// TIA Portal V16 program export: 0 tag tables, 0 data types, 94 data blocks, 48 code blocks (in call order from the OBs), 0 instance data blocks

DATA_BLOCK "DBl_SCALE_CS_1"
{ S7_Optimized_Access := 'FALSE' }
VERSION : 0.1
   STRUCT 
      Data { S7_SetPoint := 'False'} : "UDT_SIWA_CS";
   END_STRUCT;


BEGIN

END_DATA_BLOCK

DATA_BLOCK "DBl_SCALE_CS_2"
{ S7_Optimized_Access := 'FALSE' }
VERSION : 0.1
   STRUCT 
      Data { S7_SetPoint := 'False'} : "UDT_SIWA_CS";
   END_STRUCT;


BEGIN

END_DATA_BLOCK

DATA_BLOCK "DB_DateTime"
{ S7_Optimized_Access := 'FALSE' }
VERSION : 0.1
NON_RETAIN
   STRUCT 
      TimeOfDay_PLC : Time_Of_Day;
      Date_PLC : Date;
      DateTime_PLC : Date_And_Time;
      stReadDataTime_PLC : Int;
   END_STRUCT;


BEGIN
   TimeOfDay_PLC := TOD#16:14:12.371;
   Date_PLC := D#2021-11-15;
   DateTime_PLC := DT#2021-11-15-16:14:12.374;
   stReadDataTime_PLC := 0;

END_DATA_BLOCK

DATA_BLOCK "DB_Global"
{ S7_Optimized_Access := 'FALSE' }
VERSION : 0.1
NON_RETAIN
// 2. GLOBAL DATA (Pure Data only)
   STRUCT 
      Sys { ExternalAccessible := 'False'; ExternalVisible := 'False'; ExternalWritable := 'False'; S7_SetPoint := 'False'} : "UDT_Sys_Info";
      c_stDI_Mode { ExternalAccessible := 'False'; ExternalVisible := 'False'; ExternalWritable := 'False'} : Struct
         None { ExternalAccessible := 'False'; ExternalVisible := 'False'; ExternalWritable := 'False'} : Int;
         NOpen { ExternalAccessible := 'False'; ExternalVisible := 'False'; ExternalWritable := 'False'} : Int;
         NClose { ExternalAccessible := 'False'; ExternalVisible := 'False'; ExternalWritable := 'False'} : Int;
         Disabled { ExternalAccessible := 'False'; ExternalVisible := 'False'; ExternalWritable := 'False'} : Int;
      END_STRUCT;
   END_STRUCT;


BEGIN
   Sys.CycleTime_ms_INT := 10;
   Sys.CycleTime_ms_REAL := 10.0;
   c_stDI_Mode.NOpen := 1;
   c_stDI_Mode.NClose := 2;
   c_stDI_Mode.Disabled := 3;

END_DATA_BLOCK

DATA_BLOCK "DB_Log_Buffer"
{ S7_Optimized_Access := 'FALSE' }
VERSION : 0.1
   STRUCT 
      Write_Index : Int;   // Указатель для ПЛК (куда пишем следующую запись)
      Read_Index : Int;   // Указатель для Python/1C (что считано)
      Buffer : Array[0..1999] of "UDT_Log_Record";   // Кольцевой буфер на 500 записей
   END_STRUCT;


BEGIN
   Write_Index := 0;
   Read_Index := 0;

END_DATA_BLOCK

DATA_BLOCK "DB_MAP"
{ S7_Optimized_Access := 'FALSE' }
VERSION : 0.1
NON_RETAIN
   STRUCT 
      HMI_Whouse : Struct
         TRN { S7_SetPoint := 'False'} : "UDT_HMI_Whouse";
         POL { S7_SetPoint := 'False'} : "UDT_HMI_Whouse";
         BUL { S7_SetPoint := 'False'} : "UDT_HMI_Whouse";
         MOL { S7_SetPoint := 'False'} : "UDT_HMI_Whouse";
      END_STRUCT;
      HMI_TRN_SmalTank { S7_SetPoint := 'False'} : Array[1..3] of "UDT_HMI_SmallTank";
      HMI_POL_SmalTank { S7_SetPoint := 'False'} : Array[1..10] of "UDT_HMI_SmallTank";
      HMI_BUL_SmalTank { S7_SetPoint := 'False'} : Array[1..4] of "UDT_HMI_SmallTank";
      HMI_MOL_SmalTank { S7_SetPoint := 'False'} : Array[1..12] of "UDT_HMI_SmallTank";
      Scale_CS_1 : "UDT_Siwarex_Core";
      Scale_CS_2 : "UDT_Siwarex_Core";
   END_STRUCT;


BEGIN

END_DATA_BLOCK

DATA_BLOCK "DB_Wh_BUL"
{ S7_Optimized_Access := 'FALSE' }
VERSION : 0.1
   STRUCT 
      Tank : Array[1..4] of "UDT_Tank_Full";
   END_STRUCT;


BEGIN

END_DATA_BLOCK

DATA_BLOCK "DB_Wh_MOL"
{ S7_Optimized_Access := 'FALSE' }
VERSION : 0.1
   STRUCT 
      Tank : Array[1..10] of "UDT_Tank_Full";
   END_STRUCT;


BEGIN

END_DATA_BLOCK

DATA_BLOCK "DB_Wh_POL"
{ S7_Optimized_Access := 'FALSE' }
VERSION : 0.1
   STRUCT 
      Tank : Array[1..10] of "UDT_Tank_Full";
   END_STRUCT;


BEGIN

END_DATA_BLOCK

DATA_BLOCK "DB_Wh_TRN"
{ S7_Optimized_Access := 'FALSE' }
VERSION : 0.1
   STRUCT 
      HMI_Word_spare : DWord;
      Tank : Array[1..3] of "UDT_Tank_Full";
   END_STRUCT;


BEGIN

END_DATA_BLOCK

DATA_BLOCK "Total_DB"
{ S7_Optimized_Access := 'FALSE' }
VERSION : 0.1
NON_RETAIN
   STRUCT 
      Total_Reset_HMI : Bool;
      Restart_PLC : Bool;
   END_STRUCT;


BEGIN
   Total_Reset_HMI := FALSE;
   Restart_PLC := FALSE;

END_DATA_BLOCK

DATA_BLOCK "iDB_BUL_Tank_Log_1"
{ S7_Optimized_Access := 'FALSE' }
AUTHOR : Gemini
FAMILY : Archive
VERSION : 1.2
NON_RETAIN
"FB_Tank_Logic"

BEGIN

END_DATA_BLOCK

DATA_BLOCK "iDB_BUL_Tank_Log_2"
{ S7_Optimized_Access := 'FALSE' }
AUTHOR : Gemini
FAMILY : Archive
VERSION : 1.2
NON_RETAIN
"FB_Tank_Logic"

BEGIN

END_DATA_BLOCK

DATA_BLOCK "iDB_BUL_Tank_Log_3"
{ S7_Optimized_Access := 'FALSE' }
AUTHOR : Gemini
FAMILY : Archive
VERSION : 1.2
NON_RETAIN
"FB_Tank_Logic"

BEGIN

END_DATA_BLOCK

DATA_BLOCK "iDB_BUL_Tank_Log_4"
{ S7_Optimized_Access := 'FALSE' }
AUTHOR : Gemini
FAMILY : Archive
VERSION : 1.2
NON_RETAIN
"FB_Tank_Logic"

BEGIN

END_DATA_BLOCK

DATA_BLOCK "iDB_MOL_Tank_Log_1"
{ S7_Optimized_Access := 'FALSE' }
AUTHOR : Gemini
FAMILY : Archive
VERSION : 1.2
NON_RETAIN
"FB_Tank_Logic"

BEGIN

END_DATA_BLOCK

DATA_BLOCK "iDB_MOL_Tank_Log_10"
{ S7_Optimized_Access := 'FALSE' }
AUTHOR : Gemini
FAMILY : Archive
VERSION : 1.2
NON_RETAIN
"FB_Tank_Logic"

BEGIN

END_DATA_BLOCK

DATA_BLOCK "iDB_MOL_Tank_Log_11"
{ S7_Optimized_Access := 'FALSE' }
AUTHOR : Gemini
FAMILY : Archive
VERSION : 1.2
NON_RETAIN
"FB_Tank_Logic"

BEGIN

END_DATA_BLOCK

DATA_BLOCK "iDB_MOL_Tank_Log_12"
{ S7_Optimized_Access := 'FALSE' }
AUTHOR : Gemini
FAMILY : Archive
VERSION : 1.2
NON_RETAIN
"FB_Tank_Logic"

BEGIN

END_DATA_BLOCK

DATA_BLOCK "iDB_MOL_Tank_Log_2"
{ S7_Optimized_Access := 'FALSE' }
AUTHOR : Gemini
FAMILY : Archive
VERSION : 1.2
NON_RETAIN
"FB_Tank_Logic"

BEGIN

END_DATA_BLOCK

DATA_BLOCK "iDB_MOL_Tank_Log_3"
{ S7_Optimized_Access := 'FALSE' }
AUTHOR : Gemini
FAMILY : Archive
VERSION : 1.2
NON_RETAIN
"FB_Tank_Logic"

BEGIN

END_DATA_BLOCK

DATA_BLOCK "iDB_MOL_Tank_Log_4"
{ S7_Optimized_Access := 'FALSE' }
AUTHOR : Gemini
FAMILY : Archive
VERSION : 1.2
NON_RETAIN
"FB_Tank_Logic"

BEGIN

END_DATA_BLOCK

DATA_BLOCK "iDB_MOL_Tank_Log_5"
{ S7_Optimized_Access := 'FALSE' }
AUTHOR : Gemini
FAMILY : Archive
VERSION : 1.2
NON_RETAIN
"FB_Tank_Logic"

BEGIN

END_DATA_BLOCK

DATA_BLOCK "iDB_MOL_Tank_Log_6"
{ S7_Optimized_Access := 'FALSE' }
AUTHOR : Gemini
FAMILY : Archive
VERSION : 1.2
NON_RETAIN
"FB_Tank_Logic"

BEGIN

END_DATA_BLOCK

DATA_BLOCK "iDB_MOL_Tank_Log_7"
{ S7_Optimized_Access := 'FALSE' }
AUTHOR : Gemini
FAMILY : Archive
VERSION : 1.2
NON_RETAIN
"FB_Tank_Logic"

BEGIN

END_DATA_BLOCK

DATA_BLOCK "iDB_MOL_Tank_Log_8"
{ S7_Optimized_Access := 'FALSE' }
AUTHOR : Gemini
FAMILY : Archive
VERSION : 1.2
NON_RETAIN
"FB_Tank_Logic"

BEGIN

END_DATA_BLOCK

DATA_BLOCK "iDB_MOL_Tank_Log_9"
{ S7_Optimized_Access := 'FALSE' }
AUTHOR : Gemini
FAMILY : Archive
VERSION : 1.2
NON_RETAIN
"FB_Tank_Logic"

BEGIN

END_DATA_BLOCK

DATA_BLOCK "iDB_POL_Tank_Log_1"
{ S7_Optimized_Access := 'FALSE' }
AUTHOR : Gemini
FAMILY : Archive
VERSION : 1.2
"FB_Tank_Logic"

BEGIN

END_DATA_BLOCK

DATA_BLOCK "iDB_POL_Tank_Log_10"
{ S7_Optimized_Access := 'FALSE' }
AUTHOR : Gemini
FAMILY : Archive
VERSION : 1.2
NON_RETAIN
"FB_Tank_Logic"

BEGIN

END_DATA_BLOCK

DATA_BLOCK "iDB_POL_Tank_Log_3"
{ S7_Optimized_Access := 'FALSE' }
AUTHOR : Gemini
FAMILY : Archive
VERSION : 1.2
"FB_Tank_Logic"

BEGIN

END_DATA_BLOCK

DATA_BLOCK "iDB_POL_Tank_Log_4"
{ S7_Optimized_Access := 'FALSE' }
AUTHOR : Gemini
FAMILY : Archive
VERSION : 1.2
"FB_Tank_Logic"

BEGIN

END_DATA_BLOCK

DATA_BLOCK "iDB_POL_Tank_Log_5"
{ S7_Optimized_Access := 'FALSE' }
AUTHOR : Gemini
FAMILY : Archive
VERSION : 1.2
"FB_Tank_Logic"

BEGIN

END_DATA_BLOCK

DATA_BLOCK "iDB_POL_Tank_Log_6"
{ S7_Optimized_Access := 'FALSE' }
AUTHOR : Gemini
FAMILY : Archive
VERSION : 1.2
"FB_Tank_Logic"

BEGIN

END_DATA_BLOCK

DATA_BLOCK "iDB_POL_Tank_Log_7"
{ S7_Optimized_Access := 'FALSE' }
AUTHOR : Gemini
FAMILY : Archive
VERSION : 1.2
NON_RETAIN
"FB_Tank_Logic"

BEGIN

END_DATA_BLOCK

DATA_BLOCK "iDB_POL_Tank_Log_8"
{ S7_Optimized_Access := 'FALSE' }
AUTHOR : Gemini
FAMILY : Archive
VERSION : 1.2
NON_RETAIN
"FB_Tank_Logic"

BEGIN

END_DATA_BLOCK

DATA_BLOCK "iDB_POL_Tank_Log_9"
{ S7_Optimized_Access := 'FALSE' }
AUTHOR : Gemini
FAMILY : Archive
VERSION : 1.2
NON_RETAIN
"FB_Tank_Logic"

BEGIN

END_DATA_BLOCK

DATA_BLOCK "iDB_TRN_Tank_Log_1"
{ S7_Optimized_Access := 'FALSE' }
AUTHOR : Gemini
FAMILY : Archive
VERSION : 1.2
NON_RETAIN
"FB_Tank_Logic"

BEGIN

END_DATA_BLOCK

DATA_BLOCK "iDB_TRN_Tank_Log_2"
{ S7_Optimized_Access := 'FALSE' }
AUTHOR : Gemini
FAMILY : Archive
VERSION : 1.2
NON_RETAIN
"FB_Tank_Logic"

BEGIN

END_DATA_BLOCK

DATA_BLOCK "iDB_TRN_Tank_Log_3"
{ S7_Optimized_Access := 'FALSE' }
AUTHOR : Gemini
FAMILY : Archive
VERSION : 1.2
NON_RETAIN
"FB_Tank_Logic"

BEGIN

END_DATA_BLOCK

DATA_BLOCK "iDB_Time_Trigger"
{ S7_Optimized_Access := 'FALSE' }
AUTHOR : S7A_Lib
FAMILY : Archive
VERSION : 1.1
"FB_Time_Trigger"

BEGIN

END_DATA_BLOCK

DATA_BLOCK "Pol_sklad_db"
{ S7_Optimized_Access := 'FALSE' }
VERSION : 0.1
   STRUCT 
      Pol_p : Real;
      Eror_pol_p : DWord;
      S_pol : Real;
      Weigt : Real;
      Densyty : Real;
      "1_pol" : Struct
         Weight_db : Real;
         Weight_zero : Real;
         Weight_Formula_W_T : Real;
         Visible : Bool;
         p_zero : Real;
         p_weight : Real;
         Zero_but : Bool;
         Weight_but : Bool;
         S : Real;
         Densyty : Real;
         Korect : Bool;
      END_STRUCT;
      "2_pol" : Struct
         Weight_db : Real;
         Weight_zero : Real;
         Weight_Formula_W_T : Real;
         Visible : Bool;
         p_zero : Real;
         p_weight : Real;
         Zero_but : Bool;
         Weight_but : Bool;
         S : Real;
         Densyty : Real;
         Korect : Bool;
      END_STRUCT;
      "3_pol" : Struct
         Weight_db : Real;
         Weight_zero : Real;
         Weight_Formula_W_T : Real;
         Visible : Bool;
         p_zero : Real;
         p_weight : Real;
         Zero_but : Bool;
         Weight_but : Bool;
         S : Real;
         Densyty : Real;
         Korect : Bool;
      END_STRUCT;
      "4_pol" : Struct
         Weight_db : Real;
         Weight_zero : Real;
         Weight_Formula_W_T : Real;
         Visible : Bool;
         p_zero : Real;
         p_weight : Real;
         Zero_but : Bool;
         Weight_but : Bool;
         S : Real;
         Densyty : Real;
         Korect : Bool;
      END_STRUCT;
      "5_pol" : Struct
         Weight_db : Real;
         Weight_zero : Real;
         Weight_Formula_W_T : Real;
         Visible : Bool;
         p_zero : Real;
         p_weight : Real;
         Zero_but : Bool;
         Weight_but : Bool;
         S : Real;
         Densyty : Real;
         Korect : Bool;
      END_STRUCT;
      "6_pol" : Struct
         Weight_db : Real;
         Weight_zero : Real;
         Weight_Formula_W_T : Real;
         Visible : Bool;
         p_zero : Real;
         p_weight : Real;
         Zero_but : Bool;
         Weight_but : Bool;
         S : Real;
         Densyty : Real;
         Korect : Bool;
      END_STRUCT;
      "7_pol" : Struct
         Weight_db : Real;
         Weight_zero : Real;
         Weight_Formula_W_T : Real;
         Visible : Bool;
         p_zero : Real;
         p_weight : Real;
         Zero_but : Bool;
         Weight_but : Bool;
         S : Real;
         Densyty : Real;
         Korect : Bool;
      END_STRUCT;
      "8_pol" : Struct
         Weight_db : Real;
         Weight_zero : Real;
         Weight_Formula_W_T : Real;
         Visible : Bool;
         p_zero : Real;
         p_weight : Real;
         Zero_but : Bool;
         Weight_but : Bool;
         S : Real;
         Densyty : Real;
         Korect : Bool;
      END_STRUCT;
      "9_pol" : Struct
         Weight_db : Real;
         Weight_zero : Real;
         Weight_Formula_W_T : Real;
         Visible : Bool;
         p_zero : Real;
         p_weight : Real;
         Zero_but : Bool;
         Weight_but : Bool;
         S : Real;
         Densyty : Real;
         Korect : Bool;
      END_STRUCT;
      "10_pol" : Struct
         Weight_db : Real;
         Weight_zero : Real;
         Weight_Formula_W_T : Real;
         Visible : Bool;
         p_zero : Real;
         p_weight : Real;
         Zero_but : Bool;
         Weight_but : Bool;
         S : Real;
         Densyty : Real;
         Korect : Bool;
      END_STRUCT;
   END_STRUCT;


BEGIN
   Pol_p := 1.149812;
   Eror_pol_p := 16#0000_0000;
   S_pol := 6.819987;
   Weigt := 79.9358;
   Densyty := 1.35;
   "1_pol".Weight_db := 0.0;
   "1_pol".Weight_zero := 0.0;
   "1_pol".Weight_Formula_W_T := 81.81128;
   "1_pol".Visible := TRUE;
   "1_pol".p_zero := 0.0;
   "1_pol".p_weight := 0.0;
   "1_pol".Zero_but := FALSE;
   "1_pol".Weight_but := FALSE;
   "1_pol".S := 6.98;
   "1_pol".Densyty := 1.35;
   "1_pol".Korect := FALSE;
   "2_pol".Weight_db := 19.52373;
   "2_pol".Weight_zero := 0.0;
   "2_pol".Weight_Formula_W_T := 78.76387;
   "2_pol".Visible := FALSE;
   "2_pol".p_zero := 0.0;
   "2_pol".p_weight := 0.2850116;
   "2_pol".Zero_but := FALSE;
   "2_pol".Weight_but := FALSE;
   "2_pol".S := 6.72;
   "2_pol".Densyty := 1.35;
   "2_pol".Korect := FALSE;
   "3_pol".Weight_db := 0.0;
   "3_pol".Weight_zero := 0.0;
   "3_pol".Weight_Formula_W_T := 78.52945;
   "3_pol".Visible := FALSE;
   "3_pol".p_zero := 0.0;
   "3_pol".p_weight := 0.0;
   "3_pol".Zero_but := FALSE;
   "3_pol".Weight_but := FALSE;
   "3_pol".S := 6.7;
   "3_pol".Densyty := 1.35;
   "3_pol".Korect := FALSE;
   "4_pol".Weight_db := 73.68473;
   "4_pol".Weight_zero := 0.0;
   "4_pol".Weight_Formula_W_T := 78.76387;
   "4_pol".Visible := FALSE;
   "4_pol".p_zero := 0.0;
   "4_pol".p_weight := 1.075665;
   "4_pol".Zero_but := FALSE;
   "4_pol".Weight_but := FALSE;
   "4_pol".S := 6.72;
   "4_pol".Densyty := 1.35;
   "4_pol".Korect := FALSE;
   "5_pol".Weight_db := 24.61529;
   "5_pol".Weight_zero := 0.0;
   "5_pol".Weight_Formula_W_T := 77.55404;
   "5_pol".Visible := FALSE;
   "5_pol".p_zero := 0.0;
   "5_pol".p_weight := 0.364945;
   "5_pol".Zero_but := FALSE;
   "5_pol".Weight_but := FALSE;
   "5_pol".S := 6.61678;
   "5_pol".Densyty := 1.35;
   "5_pol".Korect := FALSE;
   "6_pol".Weight_db := 49.182;
   "6_pol".Weight_zero := 0.0;
   "6_pol".Weight_Formula_W_T := 78.64666;
   "6_pol".Visible := FALSE;
   "6_pol".p_zero := 0.0;
   "6_pol".p_weight := 0.7190394;
   "6_pol".Zero_but := FALSE;
   "6_pol".Weight_but := FALSE;
   "6_pol".S := 6.71;
   "6_pol".Densyty := 1.35;
   "6_pol".Korect := FALSE;
   "7_pol".Weight_db := 123.4003;
   "7_pol".Weight_zero := 0.0;
   "7_pol".Weight_Formula_W_T := 78.64666;
   "7_pol".Visible := FALSE;
   "7_pol".p_zero := 0.0;
   "7_pol".p_weight := 1.804109;
   "7_pol".Zero_but := FALSE;
   "7_pol".Weight_but := FALSE;
   "7_pol".S := 6.71;
   "7_pol".Densyty := 1.35;
   "7_pol".Korect := FALSE;
   "8_pol".Weight_db := -0.2724785;
   "8_pol".Weight_zero := 0.4211032;
   "8_pol".Weight_Formula_W_T := 78.74628;
   "8_pol".Visible := FALSE;
   "8_pol".p_zero := 0.006148727;
   "8_pol".p_weight := 0.002170139;
   "8_pol".Zero_but := FALSE;
   "8_pol".Weight_but := FALSE;
   "8_pol".S := 6.7185;
   "8_pol".Densyty := 1.35;
   "8_pol".Korect := FALSE;
   "9_pol".Weight_db := 126.8467;
   "9_pol".Weight_zero := 0.0;
   "9_pol".Weight_Formula_W_T := 78.97484;
   "9_pol".Visible := FALSE;
   "9_pol".p_zero := 0.0;
   "9_pol".p_weight := 1.846788;
   "9_pol".Zero_but := FALSE;
   "9_pol".Weight_but := FALSE;
   "9_pol".S := 6.738;
   "9_pol".Densyty := 1.35;
   "9_pol".Korect := FALSE;
   "10_pol".Weight_db := 27.88432;
   "10_pol".Weight_zero := 0.0;
   "10_pol".Weight_Formula_W_T := 77.55404;
   "10_pol".Visible := TRUE;
   "10_pol".p_zero := 0.0;
   "10_pol".p_weight := 0.4134114;
   "10_pol".Zero_but := FALSE;
   "10_pol".Weight_but := FALSE;
   "10_pol".S := 6.61678;
   "10_pol".Densyty := 1.35;
   "10_pol".Korect := FALSE;

END_DATA_BLOCK

DATA_BLOCK "iDB_Map_Siwarex_Core"
{ S7_Optimized_Access := 'FALSE' }
AUTHOR : S7C_Lib
FAMILY : Analog
VERSION : 1.4
"FB_Map_Siwarex_Core"

BEGIN

END_DATA_BLOCK

DATA_BLOCK "iFB_Map_Siwarex_Core"
{ S7_Optimized_Access := 'FALSE' }
AUTHOR : S7C_Lib
FAMILY : Analog
VERSION : 1.4
"FB_Map_Siwarex_Core"

BEGIN

END_DATA_BLOCK

DATA_BLOCK "MaxLevels"
{ S7_Optimized_Access := 'FALSE' }
VERSION : 0.1
   STRUCT 
      MaxLevel_Tank_1 : Real;
      MaxLevel_Tank_2 : Real;
      MaxLevel_Tank_3 : Real;
      MaxLevel_Tank_4 : Real;
      MaxLevel_Tank_5 : Real;
      MaxLevel_Tank_6 : Real;
      MaxLevel_Tank_7 : Real;
      MaxLevel_Tank_8 : Real;
      MaxLevel_Tank_9 : Real;
      MaxLevel_Tank_10 : Real;
      MaxLevel_Tank_11 : Real;
      MaxLevel_Tank_12 : Real;
      MaxLevel_Tank_13 : Real;
      MaxLevel_Tank_14 : Real;
   END_STRUCT;


BEGIN
   MaxLevel_Tank_1 := 15.0;
   MaxLevel_Tank_2 := 15.0;
   MaxLevel_Tank_3 := 15.0;
   MaxLevel_Tank_4 := 15.0;
   MaxLevel_Tank_5 := 15.0;
   MaxLevel_Tank_6 := 15.0;
   MaxLevel_Tank_7 := 15.0;
   MaxLevel_Tank_8 := 15.0;
   MaxLevel_Tank_9 := 15.0;
   MaxLevel_Tank_10 := 15.0;
   MaxLevel_Tank_11 := 13.0;
   MaxLevel_Tank_12 := 13.0;
   MaxLevel_Tank_13 := 13.0;
   MaxLevel_Tank_14 := 13.0;

END_DATA_BLOCK

DATA_BLOCK "DB_SCALE_CS_1"
{ S7_Optimized_Access := 'FALSE' }
VERSION : 0.0
"UDT_SIWA_CS"

BEGIN
   i_DB_Lenght := 222;
   i_MaxLifeBitCyc := 500;
   i_SFC_ERR_C := 16#0000;
   i_CMD_INPUT := 230;
   bo_CMD_TRIGGER := TRUE;
   bo_CMD_IN_PROGRESS := TRUE;
   bo_CMD_FINISHED_OK := FALSE;
   bo_CMD_ERR := FALSE;
   b_CMD_ERR_CODE := 16#00;
   i_PRESET_TARE := 0;
   b_SELECT_PROC_VAL := 16#00;
   b_SELECTED_PROC_VAL := 16#00;
   i_PROCESS_VALUE := 215;
   b_INFO_REFRESH_COUNT := 16#5A;
   w_SCALE_STATUS := 16#00C0;
   b_OPR_ERR_MSG := 16#00;
   bo_FB_ERR := FALSE;
   b_FB_ERR_CODE := 16#00;
   bo_START_UP_IN_PROGRESS := FALSE;
   w_DB_RES92 := 16#0000;
   w_DB_RES93 := 16#0000;
   w_DB_RES94 := 16#0000;
   w_DB_RES95 := 16#0000;
   w_DB_RES96 := 16#0000;
   w_DB_RES97 := 16#0000;
   w_INT_USE := 16#0000;
   s_JUST_DAT.w_CALIB_DIGITS0 := 16#0000;
   s_JUST_DAT.w_CALIB_DIGITS1 := 16#EA60;
   s_JUST_DAT.w_CALIB_DIGITS2 := 16#0000;
   s_JUST_DAT.i_CALIB_WEIGHT1 := 2000;
   s_JUST_DAT.i_CALIB_WEIGHT2 := 0;
   s_JUST_DAT.b_SIGNAL_RANGE := 16#02;
   s_JUST_DAT.b_FILT_TYPE := 16#00;
   s_JUST_DAT.b_FILT_FREQ := 16#04;
   s_JUST_DAT.b_FILT_DEPTH := 16#0F;
   s_JUST_DAT.s_SCALE_ID := 'SIWAREX XX';
   s_JUST_DAT.i_MIN_WR := 20;
   s_JUST_DAT.i_MAX_WR := 2000;
   s_JUST_DAT.i_INCREMENT_WR := 1;
   s_JUST_DAT.i_WEIGHT_ST_STILL := 10;
   s_JUST_DAT.t_TIME_ST_STILL1 := T#1S;
   s_JUST_DAT.b_DEC_POINT := 16#02;
   s_JUST_DAT.b_ZERO_NEG_VALUE := 16#01;
   s_JUST_DAT.b_ZERO_POS_VALUE := 16#03;
   s_JUST_DAT.b_TARA_MAX := 16#64;
   s_JUST_DAT.i_Reserve := 0;
   s_JUST_DAT.s_LEGAL_TRADE := '----';
   s_JUST_DAT.s_WEGHT_UNIT := 'kg  ';
   s_LIMIT_PARA.i_LIMIT1_ON := 400;
   s_LIMIT_PARA.i_LIMIT1_OFF := 220;
   s_LIMIT_PARA.i_LIMIT2_ON := 1000;
   s_LIMIT_PARA.i_LIMIT2_OFF := 980;
   s_LIMIT_PARA.bo_LIMIT1_PARA := FALSE;
   s_LIMIT_PARA.bo_LIMIT2_PARA := FALSE;
   s_LIMIT_PARA.b_Reserve := 16#00;
   s_MODUL_INFO_DATA.s_MODUL_NAME := 'SIWAREX CS';
   s_MODUL_INFO_DATA.s_ORDER_NUM := '7MH4910-0AA01$00$00$00$00   ';
   s_MODUL_INFO_DATA.w_VERSION_HW := 16#0005;
   s_MODUL_INFO_DATA.s_VERSION_FW := 'V1.5';
   s_MODUL_INFO_DATA.w_CRC_CHECK := 16#0897;
   s_TARE_CONTROL.i_TARE_VALUE := 0;
   s_INTERNAL_PROC_VAL.w_CRC_CHECK := 16#0000;
   s_INTERNAL_PROC_VAL.b_Reserve := 16#00;
   s_INTERNAL_PROC_VAL.bo_PRESET_TARA := FALSE;
   s_INTERNAL_PROC_VAL.d_TARA_X_100 := 0;
   s_INTERNAL_PROC_VAL.d_ZERO_X_100 := 0;
   s_PROCESS_VALUES.w_CRC_CHECK := 16#4732;
   s_PROCESS_VALUES.bo_STA_WRI_PROT := FALSE;
   s_PROCESS_VALUES.bo_STA_WR_MIN := FALSE;
   s_PROCESS_VALUES.bo_STA_Reserve1 := FALSE;
   s_PROCESS_VALUES.bo_STA_Reserve2 := FALSE;
   s_PROCESS_VALUES.bo_STA_Reserve3 := FALSE;
   s_PROCESS_VALUES.bo_STA_Reserve4 := FALSE;
   s_PROCESS_VALUES.bo_STA_Reserve5 := FALSE;
   s_PROCESS_VALUES.bo_STA_ERROR_ON := FALSE;
   s_PROCESS_VALUES.bo_STA_LIMIT1_ON := FALSE;
   s_PROCESS_VALUES.bo_STA_LIMIT2_ON := FALSE;
   s_PROCESS_VALUES.bo_STA_TARED := FALSE;
   s_PROCESS_VALUES.bo_STA_TARED_BY_MANUAL := FALSE;
   s_PROCESS_VALUES.bo_STA_MAX_9E := FALSE;
   s_PROCESS_VALUES.bo_STA_025_D_ZERO := FALSE;
   s_PROCESS_VALUES.bo_STA_ST_STAND_SCALE_ON := TRUE;
   s_PROCESS_VALUES.bo_STA_SCALE_CALIBRATED := TRUE;
   s_PROCESS_VALUES.b_OPR_ERR_MSG := 16#00;
   s_PROCESS_VALUES.b_Reserve := 16#00;
   s_PROCESS_VALUES.i_GROSS_WEIGHT_PROC := 217;
   s_PROCESS_VALUES.i_NET_WEIGHT_PROC := 217;
   s_PROCESS_VALUES.i_TARE_WEIGHT_PROC := 0;
   s_PROCESS_VALUES.i_GROSS_NET_VALUE := 215;
   s_PROCESS_VALUES.d_GROSS_NET_VALUE_10X := 2175;
   s_PROCESS_VALUES.i_TARE_VALUE := 0;
   s_PROCESS_VALUES.i_ADC_DIGIT := 8980;
   s_PROCESS_VALUES.i_ADC_DIGIT_FILTER := 8982;
   s_PROCESS_VALUES.s_WEIGHT_ASCII := 'B      215kg  ';
   s_PROCESS_VALUES.i_MILISEC := 180;
   s_PROCESS_VALUES.b_SECONDS := 16#2A;
   s_PROCESS_VALUES.b_MINUTE := 16#39;
   s_PROCESS_VALUES.i_HOURS := 57;
   i_DB_Lenght1 := 222;

END_DATA_BLOCK

DATA_BLOCK "DB_SCALE_CS_2"
{ S7_Optimized_Access := 'FALSE' }
VERSION : 0.0
"UDT_SIWA_CS"

BEGIN
   i_DB_Lenght := 222;
   i_MaxLifeBitCyc := 500;
   i_SFC_ERR_C := 16#0000;
   i_CMD_INPUT := 230;
   bo_CMD_TRIGGER := TRUE;
   bo_CMD_IN_PROGRESS := TRUE;
   bo_CMD_FINISHED_OK := FALSE;
   bo_CMD_ERR := FALSE;
   b_CMD_ERR_CODE := 16#00;
   i_PRESET_TARE := 0;
   b_SELECT_PROC_VAL := 16#00;
   b_SELECTED_PROC_VAL := 16#00;
   i_PROCESS_VALUE := -25;
   b_INFO_REFRESH_COUNT := 16#07;
   w_SCALE_STATUS := 16#02C0;
   b_OPR_ERR_MSG := 16#00;
   bo_FB_ERR := FALSE;
   b_FB_ERR_CODE := 16#00;
   bo_START_UP_IN_PROGRESS := FALSE;
   w_DB_RES92 := 16#0000;
   w_DB_RES93 := 16#0000;
   w_DB_RES94 := 16#0000;
   w_DB_RES95 := 16#0000;
   w_DB_RES96 := 16#0000;
   w_DB_RES97 := 16#0000;
   w_INT_USE := 16#0000;
   s_JUST_DAT.w_CALIB_DIGITS0 := 16#0000;
   s_JUST_DAT.w_CALIB_DIGITS1 := 16#EA60;
   s_JUST_DAT.w_CALIB_DIGITS2 := 16#0000;
   s_JUST_DAT.i_CALIB_WEIGHT1 := 2000;
   s_JUST_DAT.i_CALIB_WEIGHT2 := 0;
   s_JUST_DAT.b_SIGNAL_RANGE := 16#02;
   s_JUST_DAT.b_FILT_TYPE := 16#00;
   s_JUST_DAT.b_FILT_FREQ := 16#04;
   s_JUST_DAT.b_FILT_DEPTH := 16#0F;
   s_JUST_DAT.s_SCALE_ID := 'SIWAREX XX';
   s_JUST_DAT.i_MIN_WR := 20;
   s_JUST_DAT.i_MAX_WR := 2000;
   s_JUST_DAT.i_INCREMENT_WR := 1;
   s_JUST_DAT.i_WEIGHT_ST_STILL := 10;
   s_JUST_DAT.t_TIME_ST_STILL1 := T#1S;
   s_JUST_DAT.b_DEC_POINT := 16#02;
   s_JUST_DAT.b_ZERO_NEG_VALUE := 16#01;
   s_JUST_DAT.b_ZERO_POS_VALUE := 16#03;
   s_JUST_DAT.b_TARA_MAX := 16#64;
   s_JUST_DAT.i_Reserve := 0;
   s_JUST_DAT.s_LEGAL_TRADE := '----';
   s_JUST_DAT.s_WEGHT_UNIT := 'kg  ';
   s_LIMIT_PARA.i_LIMIT1_ON := 400;
   s_LIMIT_PARA.i_LIMIT1_OFF := 220;
   s_LIMIT_PARA.i_LIMIT2_ON := 1000;
   s_LIMIT_PARA.i_LIMIT2_OFF := 980;
   s_LIMIT_PARA.bo_LIMIT1_PARA := FALSE;
   s_LIMIT_PARA.bo_LIMIT2_PARA := FALSE;
   s_LIMIT_PARA.b_Reserve := 16#00;
   s_MODUL_INFO_DATA.s_MODUL_NAME := 'SIWAREX CS';
   s_MODUL_INFO_DATA.s_ORDER_NUM := '7MH4910-0AA01$00$00$00$00   ';
   s_MODUL_INFO_DATA.w_VERSION_HW := 16#0005;
   s_MODUL_INFO_DATA.s_VERSION_FW := 'V1.5';
   s_MODUL_INFO_DATA.w_CRC_CHECK := 16#0897;
   s_TARE_CONTROL.i_TARE_VALUE := 0;
   s_INTERNAL_PROC_VAL.w_CRC_CHECK := 16#0000;
   s_INTERNAL_PROC_VAL.b_Reserve := 16#00;
   s_INTERNAL_PROC_VAL.bo_PRESET_TARA := FALSE;
   s_INTERNAL_PROC_VAL.d_TARA_X_100 := 0;
   s_INTERNAL_PROC_VAL.d_ZERO_X_100 := 0;
   s_PROCESS_VALUES.w_CRC_CHECK := 16#9561;
   s_PROCESS_VALUES.bo_STA_WRI_PROT := FALSE;
   s_PROCESS_VALUES.bo_STA_WR_MIN := TRUE;
   s_PROCESS_VALUES.bo_STA_Reserve1 := FALSE;
   s_PROCESS_VALUES.bo_STA_Reserve2 := FALSE;
   s_PROCESS_VALUES.bo_STA_Reserve3 := FALSE;
   s_PROCESS_VALUES.bo_STA_Reserve4 := FALSE;
   s_PROCESS_VALUES.bo_STA_Reserve5 := FALSE;
   s_PROCESS_VALUES.bo_STA_ERROR_ON := FALSE;
   s_PROCESS_VALUES.bo_STA_LIMIT1_ON := FALSE;
   s_PROCESS_VALUES.bo_STA_LIMIT2_ON := FALSE;
   s_PROCESS_VALUES.bo_STA_TARED := FALSE;
   s_PROCESS_VALUES.bo_STA_TARED_BY_MANUAL := FALSE;
   s_PROCESS_VALUES.bo_STA_MAX_9E := FALSE;
   s_PROCESS_VALUES.bo_STA_025_D_ZERO := FALSE;
   s_PROCESS_VALUES.bo_STA_ST_STAND_SCALE_ON := TRUE;
   s_PROCESS_VALUES.bo_STA_SCALE_CALIBRATED := TRUE;
   s_PROCESS_VALUES.b_OPR_ERR_MSG := 16#00;
   s_PROCESS_VALUES.b_Reserve := 16#00;
   s_PROCESS_VALUES.i_GROSS_WEIGHT_PROC := -27;
   s_PROCESS_VALUES.i_NET_WEIGHT_PROC := -27;
   s_PROCESS_VALUES.i_TARE_WEIGHT_PROC := 0;
   s_PROCESS_VALUES.i_GROSS_NET_VALUE := -25;
   s_PROCESS_VALUES.d_GROSS_NET_VALUE_10X := -270;
   s_PROCESS_VALUES.i_TARE_VALUE := 0;
   s_PROCESS_VALUES.i_ADC_DIGIT := 9164;
   s_PROCESS_VALUES.i_ADC_DIGIT_FILTER := 9164;
   s_PROCESS_VALUES.s_WEIGHT_ASCII := 'B -     25 kg ';
   s_PROCESS_VALUES.i_MILISEC := 520;
   s_PROCESS_VALUES.b_SECONDS := 16#33;
   s_PROCESS_VALUES.b_MINUTE := 16#39;
   s_PROCESS_VALUES.i_HOURS := 57;
   i_DB_Lenght1 := 222;

END_DATA_BLOCK

DATA_BLOCK "DB_VECTOR_CS_1"
{ S7_Optimized_Access := 'FALSE' }
VERSION : 0.1
   STRUCT 
      lenghtdb : Int;
      POS_CMD601 : Int;
      POS_CMD602 : Int;
      POS_CMD603 : Int;
      POS_CMD604 : Int;
      POS_CMD605 : Int;
      POS_CMD606 : Int;
      POS_CMD607 : Int;
      POS_CMD608 : Int;
      POS_CMD609 : Int;
      POS_CMD610 : Int;
      DR3 : Struct
         number : Byte;
         lenght : Byte;
         adress : Int;
      END_STRUCT;
      DR4 : Struct
         number : Byte;
         lenght : Byte;
         adress : Int;
      END_STRUCT;
      DR9 : Struct
         number : Byte;
         lenght : Byte;
         adress : Int;
      END_STRUCT;
      DR15 : Struct
         number : Byte;
         lenght : Byte;
         adress : Int;
      END_STRUCT;
      DR26 : Struct
         number : Byte;
         lenght : Byte;
         adress : Int;
      END_STRUCT;
      DR30 : Struct
         number : Byte;
         lenght : Byte;
         adress : Int;
      END_STRUCT;
      DR0 : Struct
         number : Byte;
         lenght : Byte;
         adress : Int;
      END_STRUCT;
      LCMD605 : Byte;
      DR1CMD605 : Byte;
      DR2CMD605 : Byte;
      DR5CMD605 : Byte;
      DR6CMD605 : Byte;
      DR11CMD605 : Byte;
      DR12CMD605 : Byte;
      CMDCMD605 : Byte;
      LCMD610 : Byte;
      DR1CMD610 : Byte;
      DR2CMD610 : Byte;
      DR5CMD610 : Byte;
      DR6CMD610 : Byte;
      CMDCMD610 : Byte;
      lendbe : Int;
   END_STRUCT;


BEGIN
   lenghtdb := 66;
   POS_CMD601 := 0;
   POS_CMD602 := 0;
   POS_CMD603 := 0;
   POS_CMD604 := 0;
   POS_CMD605 := 50;
   POS_CMD606 := 0;
   POS_CMD607 := 0;
   POS_CMD608 := 0;
   POS_CMD609 := 0;
   POS_CMD610 := 58;
   DR3.number := 16#03;
   DR3.lenght := 16#38;
   DR3.adress := 50;
   DR4.number := 16#04;
   DR4.lenght := 16#0A;
   DR4.adress := 106;
   DR9.number := 16#09;
   DR9.lenght := 16#2C;
   DR9.adress := 116;
   DR15.number := 16#0F;
   DR15.lenght := 16#02;
   DR15.adress := 160;
   DR26.number := 16#1A;
   DR26.lenght := 16#0C;
   DR26.adress := 162;
   DR30.number := 16#1E;
   DR30.lenght := 16#2E;
   DR30.adress := 174;
   DR0.number := 16#00;
   DR0.lenght := 16#00;
   DR0.adress := 0;
   LCMD605 := 16#07;
   DR1CMD605 := 16#03;
   DR2CMD605 := 16#04;
   DR5CMD605 := 16#09;
   DR6CMD605 := 16#0F;
   DR11CMD605 := 16#1A;
   DR12CMD605 := 16#1E;
   CMDCMD605 := 16#00;
   LCMD610 := 16#05;
   DR1CMD610 := 16#03;
   DR2CMD610 := 16#04;
   DR5CMD610 := 16#0F;
   DR6CMD610 := 16#1A;
   CMDCMD610 := 16#00;
   lendbe := 66;

END_DATA_BLOCK

DATA_BLOCK "DB_VECTOR_CS_2"
{ S7_Optimized_Access := 'FALSE' }
VERSION : 0.1
   STRUCT 
      lenghtdb : Int;
      POS_CMD601 : Int;
      POS_CMD602 : Int;
      POS_CMD603 : Int;
      POS_CMD604 : Int;
      POS_CMD605 : Int;
      POS_CMD606 : Int;
      POS_CMD607 : Int;
      POS_CMD608 : Int;
      POS_CMD609 : Int;
      POS_CMD610 : Int;
      DR3 : Struct
         number : Byte;
         lenght : Byte;
         adress : Int;
      END_STRUCT;
      DR4 : Struct
         number : Byte;
         lenght : Byte;
         adress : Int;
      END_STRUCT;
      DR9 : Struct
         number : Byte;
         lenght : Byte;
         adress : Int;
      END_STRUCT;
      DR15 : Struct
         number : Byte;
         lenght : Byte;
         adress : Int;
      END_STRUCT;
      DR26 : Struct
         number : Byte;
         lenght : Byte;
         adress : Int;
      END_STRUCT;
      DR30 : Struct
         number : Byte;
         lenght : Byte;
         adress : Int;
      END_STRUCT;
      DR0 : Struct
         number : Byte;
         lenght : Byte;
         adress : Int;
      END_STRUCT;
      LCMD605 : Byte;
      DR1CMD605 : Byte;
      DR2CMD605 : Byte;
      DR5CMD605 : Byte;
      DR6CMD605 : Byte;
      DR11CMD605 : Byte;
      DR12CMD605 : Byte;
      CMDCMD605 : Byte;
      LCMD610 : Byte;
      DR1CMD610 : Byte;
      DR2CMD610 : Byte;
      DR5CMD610 : Byte;
      DR6CMD610 : Byte;
      CMDCMD610 : Byte;
      lendbe : Int;
   END_STRUCT;


BEGIN
   lenghtdb := 66;
   POS_CMD601 := 0;
   POS_CMD602 := 0;
   POS_CMD603 := 0;
   POS_CMD604 := 0;
   POS_CMD605 := 50;
   POS_CMD606 := 0;
   POS_CMD607 := 0;
   POS_CMD608 := 0;
   POS_CMD609 := 0;
   POS_CMD610 := 58;
   DR3.number := 16#03;
   DR3.lenght := 16#38;
   DR3.adress := 50;
   DR4.number := 16#04;
   DR4.lenght := 16#0A;
   DR4.adress := 106;
   DR9.number := 16#09;
   DR9.lenght := 16#2C;
   DR9.adress := 116;
   DR15.number := 16#0F;
   DR15.lenght := 16#02;
   DR15.adress := 160;
   DR26.number := 16#1A;
   DR26.lenght := 16#0C;
   DR26.adress := 162;
   DR30.number := 16#1E;
   DR30.lenght := 16#2E;
   DR30.adress := 174;
   DR0.number := 16#00;
   DR0.lenght := 16#00;
   DR0.adress := 0;
   LCMD605 := 16#07;
   DR1CMD605 := 16#03;
   DR2CMD605 := 16#04;
   DR5CMD605 := 16#09;
   DR6CMD605 := 16#0F;
   DR11CMD605 := 16#1A;
   DR12CMD605 := 16#1E;
   CMDCMD605 := 16#00;
   LCMD610 := 16#05;
   DR1CMD610 := 16#03;
   DR2CMD610 := 16#04;
   DR5CMD610 := 16#0F;
   DR6CMD610 := 16#1A;
   CMDCMD610 := 16#00;
   lendbe := 66;

END_DATA_BLOCK

DATA_BLOCK "FB_SICS_DR_T1"
{ S7_Optimized_Access := 'FALSE' }
AUTHOR : AD
FAMILY : SIWAREX
NAME : SICS_DR
VERSION : 2.0
"SICS_DR"

BEGIN
   ADDR := 260;
   DB_SCALE := 21;
   DB_VECTOR := 60;
   CMD_IN := 230;
   SEL_PROC_VAL := 16#00;
   EXT_TARA := 0;
   CMD_INPR := TRUE;
   CMD_FOK := FALSE;
   CMD_ERR := FALSE;
   CMD_ERR_C := 16#00;
   REF_COUNT := 16#4A;
   ACT_SEL_PROC_VAL := 16#00;
   PROC_VAL1 := 220;
   SC_STATUS := 16#00C0;
   ERR_MSG_C := 16#00;
   FB_ERR := FALSE;
   FB_ERR_C := 16#00;
   START_UP := FALSE;
   CMD_EN := TRUE;
   sb_CMD_EN_OLD := TRUE;
   sb_DI_OLD := FALSE;
   sb_BI_OLD := FALSE;
   sb_DIQ := FALSE;
   sb_BIQ := FALSE;
   sb_LB_OLD := FALSE;
   sb_AF_OLD := FALSE;
   sb_WRITE_DS := FALSE;
   sb_SFC_ERR := FALSE;
   si_CMD_IN_NEW := 0;
   si_CMD_IN_OLD := 230;
   si_ANZ_DS := 0;
   si_NEXT_ADR := 0;
   si_LB_CNT := 1;
   sy_CMD := 16#00;
   sy_DS_NO := 16#1E;
   sw_IN := 16#004A;
   sb_CMD_ERR_C := 16#00;
   si_ADR_DS := 42;
   si_TMP_SFC_ERR_CNT := 0;
   ss_APPL_ID := 'SIWAREX CS';
   sb_APPL_ID_ERR := FALSE;
   RDREC_1.REQ := TRUE;
   RDREC_1.ID := 16#0000_0104;
   RDREC_1.INDEX := 30;
   RDREC_1.MLEN := 46;
   RDREC_1.VALID := FALSE;
   RDREC_1.BUSY := TRUE;
   RDREC_1.ERROR := FALSE;
   RDREC_1.STATUS := 16#0070_0200;
   RDREC_1.LEN := 0;
   RDREC_1.RECORD := P#DB21.DBX174.0 BYTE 46;
   WRREC_1.REQ := FALSE;
   WRREC_1.ID := 16#0000_0000;
   WRREC_1.INDEX := 0;
   WRREC_1.LEN := 0;
   WRREC_1.DONE := FALSE;
   WRREC_1.BUSY := FALSE;
   WRREC_1.ERROR := FALSE;
   WRREC_1.STATUS := 16#0000_0000;
   WRREC_1.RECORD := NULL;
   MAX_CMD_OHNE_LS := 199;
   MAX_LESE_DS := 399;
   MAX_SCHREIBE_DS := 600;
   MAX_LESE_DS_VOR_CMD := 605;
   MAX_SCHREIBE_DS_VOR_CMD := 610;
   ADR_ANZ_ZYKLEN_LIFE_BIT := 2;
   ADR_RET_VAL_SFC58_59 := 4;
   ADR_TMP_SFC_ERR_CNT := 48;
   c_CMD_ERR_ANLAUF := 16#77;
   c_CMD_ERR_C_DR_CMD := 16#11;
   c_CMD_KETTE_ABGEB := 16#00;
   c_LB_CMD_ABBRUCH := 16#00;
   c_START_DR_DB_VECTOR := 18;

END_DATA_BLOCK

DATA_BLOCK "FB_SICS_DR_T2"
{ S7_Optimized_Access := 'FALSE' }
AUTHOR : AD
FAMILY : SIWAREX
NAME : SICS_DR
VERSION : 2.2
"SICS_DR"

BEGIN
   ADDR := 280;
   DB_SCALE := 62;
   DB_VECTOR := 63;
   CMD_IN := 230;
   SEL_PROC_VAL := 16#00;
   EXT_TARA := 0;
   CMD_INPR := TRUE;
   CMD_FOK := FALSE;
   CMD_ERR := FALSE;
   CMD_ERR_C := 16#00;
   REF_COUNT := 16#01;
   ACT_SEL_PROC_VAL := 16#00;
   PROC_VAL1 := -25;
   SC_STATUS := 16#02C0;
   ERR_MSG_C := 16#00;
   FB_ERR := FALSE;
   FB_ERR_C := 16#00;
   START_UP := FALSE;
   CMD_EN := TRUE;
   sb_CMD_EN_OLD := TRUE;
   sb_DI_OLD := FALSE;
   sb_BI_OLD := FALSE;
   sb_DIQ := FALSE;
   sb_BIQ := FALSE;
   sb_LB_OLD := TRUE;
   sb_AF_OLD := FALSE;
   sb_WRITE_DS := FALSE;
   sb_SFC_ERR := FALSE;
   si_CMD_IN_NEW := 0;
   si_CMD_IN_OLD := 230;
   si_ANZ_DS := 0;
   si_NEXT_ADR := 0;
   si_LB_CNT := 1;
   sy_CMD := 16#00;
   sy_DS_NO := 16#1E;
   sw_IN := 16#0401;
   sb_CMD_ERR_C := 16#00;
   si_ADR_DS := 42;
   si_TMP_SFC_ERR_CNT := 0;
   ss_APPL_ID := 'SIWAREX CS';
   sb_APPL_ID_ERR := FALSE;
   RDREC_1.REQ := TRUE;
   RDREC_1.ID := 16#0000_0118;
   RDREC_1.INDEX := 30;
   RDREC_1.MLEN := 46;
   RDREC_1.VALID := FALSE;
   RDREC_1.BUSY := TRUE;
   RDREC_1.ERROR := FALSE;
   RDREC_1.STATUS := 16#0070_0200;
   RDREC_1.LEN := 0;
   RDREC_1.RECORD := P#DB62.DBX174.0 BYTE 46;
   WRREC_1.REQ := FALSE;
   WRREC_1.ID := 16#0000_0000;
   WRREC_1.INDEX := 0;
   WRREC_1.LEN := 0;
   WRREC_1.DONE := FALSE;
   WRREC_1.BUSY := FALSE;
   WRREC_1.ERROR := FALSE;
   WRREC_1.STATUS := 16#0000_0000;
   WRREC_1.RECORD := NULL;
   MAX_CMD_OHNE_LS := 199;
   MAX_LESE_DS := 399;
   MAX_SCHREIBE_DS := 600;
   MAX_LESE_DS_VOR_CMD := 605;
   MAX_SCHREIBE_DS_VOR_CMD := 610;
   ADR_ANZ_ZYKLEN_LIFE_BIT := 2;
   ADR_RET_VAL_SFC58_59 := 4;
   ADR_TMP_SFC_ERR_CNT := 48;
   c_CMD_ERR_ANLAUF := 16#77;
   c_CMD_ERR_C_DR_CMD := 16#11;
   c_CMD_KETTE_ABGEB := 16#00;
   c_LB_CMD_ABBRUCH := 16#00;
   c_START_DR_DB_VECTOR := 18;

END_DATA_BLOCK

DATA_BLOCK "SICS_DR_DB"
{ S7_Optimized_Access := 'FALSE' }
AUTHOR : AD
FAMILY : SIWAREX
NAME : SICS_DR
VERSION : 2.2
"SICS_DR"

BEGIN
   ADDR := 0;
   DB_SCALE := 0;
   DB_VECTOR := 0;
   CMD_IN := 0;
   SEL_PROC_VAL := 16#00;
   EXT_TARA := 0;
   CMD_INPR := FALSE;
   CMD_FOK := FALSE;
   CMD_ERR := FALSE;
   CMD_ERR_C := 16#00;
   REF_COUNT := 16#00;
   ACT_SEL_PROC_VAL := 16#00;
   PROC_VAL1 := 0;
   SC_STATUS := 16#0000;
   ERR_MSG_C := 16#00;
   FB_ERR := FALSE;
   FB_ERR_C := 16#00;
   START_UP := FALSE;
   CMD_EN := FALSE;
   sb_CMD_EN_OLD := FALSE;
   sb_DI_OLD := FALSE;
   sb_BI_OLD := FALSE;
   sb_DIQ := FALSE;
   sb_BIQ := FALSE;
   sb_LB_OLD := FALSE;
   sb_AF_OLD := FALSE;
   sb_WRITE_DS := FALSE;
   sb_SFC_ERR := FALSE;
   si_CMD_IN_NEW := 0;
   si_CMD_IN_OLD := 0;
   si_ANZ_DS := 0;
   si_NEXT_ADR := 0;
   si_LB_CNT := 0;
   sy_CMD := 16#00;
   sy_DS_NO := 16#00;
   sw_IN := 16#0000;
   sb_CMD_ERR_C := 16#00;
   si_ADR_DS := 0;
   si_TMP_SFC_ERR_CNT := 0;
   ss_APPL_ID := 'SIWAREX CS';
   sb_APPL_ID_ERR := FALSE;
   RDREC_1.REQ := FALSE;
   RDREC_1.ID := 16#0000_0000;
   RDREC_1.INDEX := 0;
   RDREC_1.MLEN := 0;
   RDREC_1.VALID := FALSE;
   RDREC_1.BUSY := FALSE;
   RDREC_1.ERROR := FALSE;
   RDREC_1.STATUS := 16#0000_0000;
   RDREC_1.LEN := 0;
   RDREC_1.RECORD := NULL;
   WRREC_1.REQ := FALSE;
   WRREC_1.ID := 16#0000_0000;
   WRREC_1.INDEX := 0;
   WRREC_1.LEN := 0;
   WRREC_1.DONE := FALSE;
   WRREC_1.BUSY := FALSE;
   WRREC_1.ERROR := FALSE;
   WRREC_1.STATUS := 16#0000_0000;
   WRREC_1.RECORD := NULL;
   MAX_CMD_OHNE_LS := 0;
   MAX_LESE_DS := 0;
   MAX_SCHREIBE_DS := 0;
   MAX_LESE_DS_VOR_CMD := 0;
   MAX_SCHREIBE_DS_VOR_CMD := 0;
   ADR_ANZ_ZYKLEN_LIFE_BIT := 0;
   ADR_RET_VAL_SFC58_59 := 0;
   ADR_TMP_SFC_ERR_CNT := 0;
   c_CMD_ERR_ANLAUF := 16#00;
   c_CMD_ERR_C_DR_CMD := 16#00;
   c_CMD_KETTE_ABGEB := 16#00;
   c_LB_CMD_ABBRUCH := 16#00;
   c_START_DR_DB_VECTOR := 0;

END_DATA_BLOCK

DATA_BLOCK "iDB_Map_Siwarex_Core_1"
{ S7_Optimized_Access := 'FALSE' }
AUTHOR : S7C_Lib
FAMILY : Analog
VERSION : 1.4
"FB_Map_Siwarex_Core"

BEGIN

END_DATA_BLOCK

DATA_BLOCK "AI_Tank1_DB"
{ S7_Optimized_Access := 'FALSE' }
AUTHOR : SimenCom
VERSION : 1.0
"Analog_In_UDT"

BEGIN

END_DATA_BLOCK

DATA_BLOCK "CalcVolume_Tank1_DB"
{ S7_Optimized_Access := 'FALSE' }
VERSION : 0.1
"CalculationVolume"

BEGIN
   IW_Radius := 1.465;
   IW_ValueFromSensor := 17.53111;
   IW_K_for_Tonnag := 1.35;
   IW_K_for_Level := 1.35;
   QW_Volume := 87.51459;
   QW_Tonnag := 118.1447;
   QW_RealLevel := 12.986;
   sW_S := 6.739147;
   sW_Volume := 87.51459;
   sW_RealLevel := 12.986;

END_DATA_BLOCK

DATA_BLOCK "UDT_AI_Tank1"
{ S7_Optimized_Access := 'FALSE' }
VERSION : 0.1
"UDT_Analog_In"

BEGIN
   IW_HW_UpLevel := 27648;
   IW_HW_LowLevel := 0;
   IDW_UpLevel := 25.0;
   IDW_LowLevel := 0.0;
   IDW_HiHi := 4.0;
   IDW_Hi := 0.0;
   IDW_Lo := 0.0;
   IDW_Lolo := 0.0;
   IW_DelayON_HiHi := 0;
   IW_DelayON_Hi := 0;
   IW_DelayON_Lo := 0;
   IW_DelayON_LoLo := 0;
   IDW_Simulation_Value := 0.0;
   IW_Time_Filter := 0;
   IW_CTW[0] := FALSE;
   IW_CTW[1] := FALSE;
   IW_CTW[2] := FALSE;
   IW_CTW[3] := FALSE;
   IW_CTW[4] := FALSE;
   IW_CTW[5] := FALSE;
   IW_CTW[6] := FALSE;
   IW_CTW[7] := FALSE;
   IW_CTW[8] := FALSE;
   IW_CTW[9] := FALSE;
   IW_CTW[10] := FALSE;
   IW_CTW[11] := FALSE;
   IW_CTW[12] := FALSE;
   IW_CTW[13] := FALSE;
   IW_CTW[14] := FALSE;
   IW_CTW[15] := FALSE;
   IDW_K_Mult := 1.0;
   IDW_DeadZone := 0.0;
   IBt_Enable_ControlLevel[0] := FALSE;
   IBt_Enable_ControlLevel[1] := FALSE;
   IBt_Enable_ControlLevel[2] := FALSE;
   IBt_Enable_ControlLevel[3] := FALSE;
   IBt_Enable_ControlLevel[4] := FALSE;
   IBt_Enable_ControlLevel[5] := FALSE;
   IBt_Enable_ControlLevel[6] := FALSE;
   IBt_Enable_ControlLevel[7] := FALSE;
   IBt_Block_ControlLevel[0] := FALSE;
   IBt_Block_ControlLevel[1] := FALSE;
   IBt_Block_ControlLevel[2] := FALSE;
   IBt_Block_ControlLevel[3] := FALSE;
   IBt_Block_ControlLevel[4] := FALSE;
   IBt_Block_ControlLevel[5] := FALSE;
   IBt_Block_ControlLevel[6] := FALSE;
   IBt_Block_ControlLevel[7] := FALSE;
   QW_STW[0] := FALSE;
   QW_STW[1] := FALSE;
   QW_STW[2] := TRUE;
   QW_STW[3] := FALSE;
   QW_STW[4] := FALSE;
   QW_STW[5] := FALSE;
   QW_STW[6] := FALSE;
   QW_STW[7] := FALSE;
   QW_STW[8] := FALSE;
   QW_STW[9] := FALSE;
   QW_STW[10] := FALSE;
   QW_STW[11] := FALSE;
   QW_STW[12] := FALSE;
   QW_STW[13] := FALSE;
   QW_STW[14] := FALSE;
   QW_STW[15] := FALSE;
   QW_HWValue := 19388;
   QDW_ScalledValue := 17.53111;
   QDW_Message[0] := FALSE;
   QDW_Message[1] := FALSE;
   QDW_Message[2] := FALSE;
   QDW_Message[3] := FALSE;
   QDW_Message[4] := FALSE;
   QDW_Message[5] := FALSE;
   QDW_Message[6] := FALSE;
   QDW_Message[7] := FALSE;
   QDW_Message[8] := FALSE;
   QDW_Message[9] := FALSE;
   QDW_Message[10] := FALSE;
   QDW_Message[11] := FALSE;
   QDW_Message[12] := FALSE;
   QDW_Message[13] := FALSE;
   QDW_Message[14] := FALSE;
   QDW_Message[15] := FALSE;
   QDW_Message[16] := FALSE;

END_DATA_BLOCK

DATA_BLOCK "AI_Tank10_DB"
{ S7_Optimized_Access := 'FALSE' }
AUTHOR : SimenCom
VERSION : 1.0
"Analog_In_UDT"

BEGIN

END_DATA_BLOCK

DATA_BLOCK "CalcVolume_Tank10_DB"
{ S7_Optimized_Access := 'FALSE' }
VERSION : 0.1
"CalculationVolume"

BEGIN
   IW_Radius := 1.468;
   IW_ValueFromSensor := 18.56192;
   IW_K_for_Tonnag := 1.35;
   IW_K_for_Level := 1.35;
   QW_Volume := 93.04028;
   QW_Tonnag := 125.6044;
   QW_RealLevel := 13.74957;
   sW_S := 6.766776;
   sW_Volume := 93.04028;
   sW_RealLevel := 13.74957;

END_DATA_BLOCK

DATA_BLOCK "UDT_AI_Tank10"
{ S7_Optimized_Access := 'FALSE' }
VERSION : 0.1
"UDT_Analog_In"

BEGIN
   IW_HW_UpLevel := 27648;
   IW_HW_LowLevel := 0;
   IDW_UpLevel := 25.0;
   IDW_LowLevel := 0.0;
   IDW_HiHi := 18.5;
   IDW_Hi := 18.0;
   IDW_Lo := 0.0;
   IDW_Lolo := 0.0;
   IW_DelayON_HiHi := 1;
   IW_DelayON_Hi := 1;
   IW_DelayON_Lo := 0;
   IW_DelayON_LoLo := 0;
   IDW_Simulation_Value := 0.0;
   IW_Time_Filter := 0;
   IW_CTW[0] := FALSE;
   IW_CTW[1] := FALSE;
   IW_CTW[2] := FALSE;
   IW_CTW[3] := FALSE;
   IW_CTW[4] := FALSE;
   IW_CTW[5] := FALSE;
   IW_CTW[6] := FALSE;
   IW_CTW[7] := FALSE;
   IW_CTW[8] := FALSE;
   IW_CTW[9] := FALSE;
   IW_CTW[10] := FALSE;
   IW_CTW[11] := FALSE;
   IW_CTW[12] := FALSE;
   IW_CTW[13] := FALSE;
   IW_CTW[14] := FALSE;
   IW_CTW[15] := FALSE;
   IDW_K_Mult := 1.0;
   IDW_DeadZone := 0.0;
   IBt_Enable_ControlLevel[0] := TRUE;
   IBt_Enable_ControlLevel[1] := TRUE;
   IBt_Enable_ControlLevel[2] := FALSE;
   IBt_Enable_ControlLevel[3] := FALSE;
   IBt_Enable_ControlLevel[4] := FALSE;
   IBt_Enable_ControlLevel[5] := FALSE;
   IBt_Enable_ControlLevel[6] := FALSE;
   IBt_Enable_ControlLevel[7] := FALSE;
   IBt_Block_ControlLevel[0] := FALSE;
   IBt_Block_ControlLevel[1] := FALSE;
   IBt_Block_ControlLevel[2] := FALSE;
   IBt_Block_ControlLevel[3] := FALSE;
   IBt_Block_ControlLevel[4] := FALSE;
   IBt_Block_ControlLevel[5] := FALSE;
   IBt_Block_ControlLevel[6] := FALSE;
   IBt_Block_ControlLevel[7] := FALSE;
   QW_STW[0] := TRUE;
   QW_STW[1] := TRUE;
   QW_STW[2] := FALSE;
   QW_STW[3] := FALSE;
   QW_STW[4] := TRUE;
   QW_STW[5] := TRUE;
   QW_STW[6] := FALSE;
   QW_STW[7] := FALSE;
   QW_STW[8] := FALSE;
   QW_STW[9] := FALSE;
   QW_STW[10] := FALSE;
   QW_STW[11] := FALSE;
   QW_STW[12] := FALSE;
   QW_STW[13] := FALSE;
   QW_STW[14] := FALSE;
   QW_STW[15] := FALSE;
   QW_HWValue := 20524;
   QDW_ScalledValue := 18.5583;
   QDW_Message[0] := FALSE;
   QDW_Message[1] := TRUE;
   QDW_Message[2] := FALSE;
   QDW_Message[3] := FALSE;
   QDW_Message[4] := FALSE;
   QDW_Message[5] := FALSE;
   QDW_Message[6] := FALSE;
   QDW_Message[7] := FALSE;
   QDW_Message[8] := FALSE;
   QDW_Message[9] := FALSE;
   QDW_Message[10] := FALSE;
   QDW_Message[11] := FALSE;
   QDW_Message[12] := FALSE;
   QDW_Message[13] := FALSE;
   QDW_Message[14] := TRUE;
   QDW_Message[15] := FALSE;
   QDW_Message[16] := FALSE;

END_DATA_BLOCK

DATA_BLOCK "AI_Tank11_DB"
{ S7_Optimized_Access := 'FALSE' }
AUTHOR : SimenCom
VERSION : 1.0
"Analog_In_UDT"

BEGIN

END_DATA_BLOCK

DATA_BLOCK "CalcVolume_Tank11_DB"
{ S7_Optimized_Access := 'FALSE' }
VERSION : 0.1
"CalculationVolume"

BEGIN
   IW_Radius := 3.102;
   IW_ValueFromSensor := 6.546586;
   IW_K_for_Tonnag := 1.35;
   IW_K_for_Level := 1.35;
   QW_Volume := 146.5191;
   QW_Tonnag := 197.8008;
   QW_RealLevel := 4.849322;
   sW_S := 30.21435;
   sW_Volume := 146.5191;
   sW_RealLevel := 4.849322;

END_DATA_BLOCK

DATA_BLOCK "UDT_AI_Tank11"
{ S7_Optimized_Access := 'FALSE' }
VERSION : 0.1
"UDT_Analog_In"

BEGIN
   IW_HW_UpLevel := 27648;
   IW_HW_LowLevel := 0;
   IDW_UpLevel := 25.0;
   IDW_LowLevel := 0.0;
   IDW_HiHi := 17.5;
   IDW_Hi := 17.0;
   IDW_Lo := 0.0;
   IDW_Lolo := 0.0;
   IW_DelayON_HiHi := 1;
   IW_DelayON_Hi := 1;
   IW_DelayON_Lo := 0;
   IW_DelayON_LoLo := 0;
   IDW_Simulation_Value := 0.0;
   IW_Time_Filter := 0;
   IW_CTW[0] := FALSE;
   IW_CTW[1] := FALSE;
   IW_CTW[2] := FALSE;
   IW_CTW[3] := FALSE;
   IW_CTW[4] := FALSE;
   IW_CTW[5] := FALSE;
   IW_CTW[6] := FALSE;
   IW_CTW[7] := FALSE;
   IW_CTW[8] := FALSE;
   IW_CTW[9] := FALSE;
   IW_CTW[10] := FALSE;
   IW_CTW[11] := FALSE;
   IW_CTW[12] := FALSE;
   IW_CTW[13] := FALSE;
   IW_CTW[14] := FALSE;
   IW_CTW[15] := FALSE;
   IDW_K_Mult := 1.0;
   IDW_DeadZone := 0.0;
   IBt_Enable_ControlLevel[0] := TRUE;
   IBt_Enable_ControlLevel[1] := TRUE;
   IBt_Enable_ControlLevel[2] := FALSE;
   IBt_Enable_ControlLevel[3] := FALSE;
   IBt_Enable_ControlLevel[4] := FALSE;
   IBt_Enable_ControlLevel[5] := FALSE;
   IBt_Enable_ControlLevel[6] := FALSE;
   IBt_Enable_ControlLevel[7] := FALSE;
   IBt_Block_ControlLevel[0] := FALSE;
   IBt_Block_ControlLevel[1] := FALSE;
   IBt_Block_ControlLevel[2] := FALSE;
   IBt_Block_ControlLevel[3] := FALSE;
   IBt_Block_ControlLevel[4] := FALSE;
   IBt_Block_ControlLevel[5] := FALSE;
   IBt_Block_ControlLevel[6] := FALSE;
   IBt_Block_ControlLevel[7] := FALSE;
   QW_STW[0] := FALSE;
   QW_STW[1] := FALSE;
   QW_STW[2] := TRUE;
   QW_STW[3] := FALSE;
   QW_STW[4] := FALSE;
   QW_STW[5] := FALSE;
   QW_STW[6] := FALSE;
   QW_STW[7] := FALSE;
   QW_STW[8] := FALSE;
   QW_STW[9] := FALSE;
   QW_STW[10] := FALSE;
   QW_STW[11] := FALSE;
   QW_STW[12] := FALSE;
   QW_STW[13] := FALSE;
   QW_STW[14] := FALSE;
   QW_STW[15] := FALSE;
   QW_HWValue := 7240;
   QDW_ScalledValue := 6.546586;
   QDW_Message[0] := FALSE;
   QDW_Message[1] := FALSE;
   QDW_Message[2] := FALSE;
   QDW_Message[3] := FALSE;
   QDW_Message[4] := FALSE;
   QDW_Message[5] := FALSE;
   QDW_Message[6] := FALSE;
   QDW_Message[7] := FALSE;
   QDW_Message[8] := FALSE;
   QDW_Message[9] := FALSE;
   QDW_Message[10] := FALSE;
   QDW_Message[11] := FALSE;
   QDW_Message[12] := FALSE;
   QDW_Message[13] := FALSE;
   QDW_Message[14] := FALSE;
   QDW_Message[15] := FALSE;
   QDW_Message[16] := FALSE;

END_DATA_BLOCK

DATA_BLOCK "AI_Tank12_DB"
{ S7_Optimized_Access := 'FALSE' }
AUTHOR : SimenCom
VERSION : 1.0
"Analog_In_UDT"

BEGIN

END_DATA_BLOCK

DATA_BLOCK "CalcVolume_Tank12_DB"
{ S7_Optimized_Access := 'FALSE' }
VERSION : 0.1
"CalculationVolume"

BEGIN
   IW_Radius := 3.102;
   IW_ValueFromSensor := 15.90712;
   IW_K_for_Tonnag := 1.35;
   IW_K_for_Level := 1.35;
   QW_Volume := 356.0172;
   QW_Tonnag := 480.6232;
   QW_RealLevel := 11.78305;
   sW_S := 30.21435;
   sW_Volume := 356.0172;
   sW_RealLevel := 11.78305;

END_DATA_BLOCK

DATA_BLOCK "UDT_AI_Tank12"
{ S7_Optimized_Access := 'FALSE' }
VERSION : 0.1
"UDT_Analog_In"

BEGIN
   IW_HW_UpLevel := 27648;
   IW_HW_LowLevel := 0;
   IDW_UpLevel := 25.0;
   IDW_LowLevel := 0.0;
   IDW_HiHi := 17.5;
   IDW_Hi := 17.0;
   IDW_Lo := 0.0;
   IDW_Lolo := 0.0;
   IW_DelayON_HiHi := 1;
   IW_DelayON_Hi := 1;
   IW_DelayON_Lo := 0;
   IW_DelayON_LoLo := 0;
   IDW_Simulation_Value := 0.0;
   IW_Time_Filter := 0;
   IW_CTW[0] := FALSE;
   IW_CTW[1] := FALSE;
   IW_CTW[2] := FALSE;
   IW_CTW[3] := FALSE;
   IW_CTW[4] := FALSE;
   IW_CTW[5] := FALSE;
   IW_CTW[6] := FALSE;
   IW_CTW[7] := FALSE;
   IW_CTW[8] := FALSE;
   IW_CTW[9] := FALSE;
   IW_CTW[10] := FALSE;
   IW_CTW[11] := FALSE;
   IW_CTW[12] := FALSE;
   IW_CTW[13] := FALSE;
   IW_CTW[14] := FALSE;
   IW_CTW[15] := FALSE;
   IDW_K_Mult := 1.0;
   IDW_DeadZone := 0.0;
   IBt_Enable_ControlLevel[0] := TRUE;
   IBt_Enable_ControlLevel[1] := TRUE;
   IBt_Enable_ControlLevel[2] := FALSE;
   IBt_Enable_ControlLevel[3] := FALSE;
   IBt_Enable_ControlLevel[4] := FALSE;
   IBt_Enable_ControlLevel[5] := FALSE;
   IBt_Enable_ControlLevel[6] := FALSE;
   IBt_Enable_ControlLevel[7] := FALSE;
   IBt_Block_ControlLevel[0] := FALSE;
   IBt_Block_ControlLevel[1] := FALSE;
   IBt_Block_ControlLevel[2] := FALSE;
   IBt_Block_ControlLevel[3] := FALSE;
   IBt_Block_ControlLevel[4] := FALSE;
   IBt_Block_ControlLevel[5] := FALSE;
   IBt_Block_ControlLevel[6] := FALSE;
   IBt_Block_ControlLevel[7] := FALSE;
   QW_STW[0] := FALSE;
   QW_STW[1] := FALSE;
   QW_STW[2] := TRUE;
   QW_STW[3] := FALSE;
   QW_STW[4] := FALSE;
   QW_STW[5] := FALSE;
   QW_STW[6] := FALSE;
   QW_STW[7] := FALSE;
   QW_STW[8] := FALSE;
   QW_STW[9] := FALSE;
   QW_STW[10] := FALSE;
   QW_STW[11] := FALSE;
   QW_STW[12] := FALSE;
   QW_STW[13] := FALSE;
   QW_STW[14] := FALSE;
   QW_STW[15] := FALSE;
   QW_HWValue := 17592;
   QDW_ScalledValue := 15.90712;
   QDW_Message[0] := FALSE;
   QDW_Message[1] := FALSE;
   QDW_Message[2] := FALSE;
   QDW_Message[3] := FALSE;
   QDW_Message[4] := FALSE;
   QDW_Message[5] := FALSE;
   QDW_Message[6] := FALSE;
   QDW_Message[7] := FALSE;
   QDW_Message[8] := FALSE;
   QDW_Message[9] := FALSE;
   QDW_Message[10] := FALSE;
   QDW_Message[11] := FALSE;
   QDW_Message[12] := FALSE;
   QDW_Message[13] := FALSE;
   QDW_Message[14] := FALSE;
   QDW_Message[15] := FALSE;
   QDW_Message[16] := FALSE;

END_DATA_BLOCK

DATA_BLOCK "AI_Tank13_DB"
{ S7_Optimized_Access := 'FALSE' }
AUTHOR : SimenCom
VERSION : 1.0
"Analog_In_UDT"

BEGIN

END_DATA_BLOCK

DATA_BLOCK "CalcVolume_Tank13_DB"
{ S7_Optimized_Access := 'FALSE' }
VERSION : 0.1
"CalculationVolume"

BEGIN
   IW_Radius := 3.102;
   IW_ValueFromSensor := 5.385561;
   IW_K_for_Tonnag := 1.35;
   IW_K_for_Level := 1.35;
   QW_Volume := 120.5342;
   QW_Tonnag := 162.7212;
   QW_RealLevel := 3.989305;
   sW_S := 30.21435;
   sW_Volume := 120.5342;
   sW_RealLevel := 3.989305;

END_DATA_BLOCK

DATA_BLOCK "UDT_AI_Tank13"
{ S7_Optimized_Access := 'FALSE' }
VERSION : 0.1
"UDT_Analog_In"

BEGIN
   IW_HW_UpLevel := 27648;
   IW_HW_LowLevel := 0;
   IDW_UpLevel := 25.0;
   IDW_LowLevel := 0.0;
   IDW_HiHi := 17.5;
   IDW_Hi := 17.0;
   IDW_Lo := 0.0;
   IDW_Lolo := 0.0;
   IW_DelayON_HiHi := 1;
   IW_DelayON_Hi := 1;
   IW_DelayON_Lo := 0;
   IW_DelayON_LoLo := 0;
   IDW_Simulation_Value := 0.0;
   IW_Time_Filter := 0;
   IW_CTW[0] := FALSE;
   IW_CTW[1] := FALSE;
   IW_CTW[2] := FALSE;
   IW_CTW[3] := FALSE;
   IW_CTW[4] := FALSE;
   IW_CTW[5] := FALSE;
   IW_CTW[6] := FALSE;
   IW_CTW[7] := FALSE;
   IW_CTW[8] := FALSE;
   IW_CTW[9] := FALSE;
   IW_CTW[10] := FALSE;
   IW_CTW[11] := FALSE;
   IW_CTW[12] := FALSE;
   IW_CTW[13] := FALSE;
   IW_CTW[14] := FALSE;
   IW_CTW[15] := FALSE;
   IDW_K_Mult := 1.0;
   IDW_DeadZone := 0.0;
   IBt_Enable_ControlLevel[0] := TRUE;
   IBt_Enable_ControlLevel[1] := TRUE;
   IBt_Enable_ControlLevel[2] := FALSE;
   IBt_Enable_ControlLevel[3] := FALSE;
   IBt_Enable_ControlLevel[4] := FALSE;
   IBt_Enable_ControlLevel[5] := FALSE;
   IBt_Enable_ControlLevel[6] := FALSE;
   IBt_Enable_ControlLevel[7] := FALSE;
   IBt_Block_ControlLevel[0] := FALSE;
   IBt_Block_ControlLevel[1] := FALSE;
   IBt_Block_ControlLevel[2] := FALSE;
   IBt_Block_ControlLevel[3] := FALSE;
   IBt_Block_ControlLevel[4] := FALSE;
   IBt_Block_ControlLevel[5] := FALSE;
   IBt_Block_ControlLevel[6] := FALSE;
   IBt_Block_ControlLevel[7] := FALSE;
   QW_STW[0] := FALSE;
   QW_STW[1] := FALSE;
   QW_STW[2] := TRUE;
   QW_STW[3] := FALSE;
   QW_STW[4] := FALSE;
   QW_STW[5] := FALSE;
   QW_STW[6] := FALSE;
   QW_STW[7] := FALSE;
   QW_STW[8] := FALSE;
   QW_STW[9] := FALSE;
   QW_STW[10] := FALSE;
   QW_STW[11] := FALSE;
   QW_STW[12] := FALSE;
   QW_STW[13] := FALSE;
   QW_STW[14] := FALSE;
   QW_STW[15] := FALSE;
   QW_HWValue := 5952;
   QDW_ScalledValue := 5.381945;
   QDW_Message[0] := FALSE;
   QDW_Message[1] := FALSE;
   QDW_Message[2] := FALSE;
   QDW_Message[3] := FALSE;
   QDW_Message[4] := FALSE;
   QDW_Message[5] := FALSE;
   QDW_Message[6] := FALSE;
   QDW_Message[7] := FALSE;
   QDW_Message[8] := FALSE;
   QDW_Message[9] := FALSE;
   QDW_Message[10] := FALSE;
   QDW_Message[11] := FALSE;
   QDW_Message[12] := FALSE;
   QDW_Message[13] := FALSE;
   QDW_Message[14] := FALSE;
   QDW_Message[15] := FALSE;
   QDW_Message[16] := FALSE;

END_DATA_BLOCK

DATA_BLOCK "AI_Tank14_DB"
{ S7_Optimized_Access := 'FALSE' }
AUTHOR : SimenCom
VERSION : 1.0
"Analog_In_UDT"

BEGIN

END_DATA_BLOCK

DATA_BLOCK "CalcVolume_Tank14_DB"
{ S7_Optimized_Access := 'FALSE' }
VERSION : 0.1
"CalculationVolume"

BEGIN
   IW_Radius := 3.102;
   IW_ValueFromSensor := 17.18027;
   IW_K_for_Tonnag := 1.35;
   IW_K_for_Level := 1.35;
   QW_Volume := 384.5115;
   QW_Tonnag := 519.0905;
   QW_RealLevel := 12.72612;
   sW_S := 30.21435;
   sW_Volume := 384.5115;
   sW_RealLevel := 12.72612;

END_DATA_BLOCK

DATA_BLOCK "UDT_AI_Tank14"
{ S7_Optimized_Access := 'FALSE' }
VERSION : 0.1
"UDT_Analog_In"

BEGIN
   IW_HW_UpLevel := 27648;
   IW_HW_LowLevel := 0;
   IDW_UpLevel := 25.0;
   IDW_LowLevel := 0.0;
   IDW_HiHi := 17.5;
   IDW_Hi := 17.0;
   IDW_Lo := 0.0;
   IDW_Lolo := 0.0;
   IW_DelayON_HiHi := 1;
   IW_DelayON_Hi := 1;
   IW_DelayON_Lo := 0;
   IW_DelayON_LoLo := 0;
   IDW_Simulation_Value := 0.0;
   IW_Time_Filter := 0;
   IW_CTW[0] := FALSE;
   IW_CTW[1] := FALSE;
   IW_CTW[2] := FALSE;
   IW_CTW[3] := FALSE;
   IW_CTW[4] := FALSE;
   IW_CTW[5] := FALSE;
   IW_CTW[6] := FALSE;
   IW_CTW[7] := FALSE;
   IW_CTW[8] := FALSE;
   IW_CTW[9] := FALSE;
   IW_CTW[10] := FALSE;
   IW_CTW[11] := FALSE;
   IW_CTW[12] := FALSE;
   IW_CTW[13] := FALSE;
   IW_CTW[14] := FALSE;
   IW_CTW[15] := FALSE;
   IDW_K_Mult := 1.0;
   IDW_DeadZone := 0.0;
   IBt_Enable_ControlLevel[0] := TRUE;
   IBt_Enable_ControlLevel[1] := TRUE;
   IBt_Enable_ControlLevel[2] := FALSE;
   IBt_Enable_ControlLevel[3] := FALSE;
   IBt_Enable_ControlLevel[4] := FALSE;
   IBt_Enable_ControlLevel[5] := FALSE;
   IBt_Enable_ControlLevel[6] := FALSE;
   IBt_Enable_ControlLevel[7] := FALSE;
   IBt_Block_ControlLevel[0] := FALSE;
   IBt_Block_ControlLevel[1] := FALSE;
   IBt_Block_ControlLevel[2] := FALSE;
   IBt_Block_ControlLevel[3] := FALSE;
   IBt_Block_ControlLevel[4] := FALSE;
   IBt_Block_ControlLevel[5] := FALSE;
   IBt_Block_ControlLevel[6] := FALSE;
   IBt_Block_ControlLevel[7] := FALSE;
   QW_STW[0] := FALSE;
   QW_STW[1] := TRUE;
   QW_STW[2] := FALSE;
   QW_STW[3] := FALSE;
   QW_STW[4] := FALSE;
   QW_STW[5] := TRUE;
   QW_STW[6] := FALSE;
   QW_STW[7] := FALSE;
   QW_STW[8] := FALSE;
   QW_STW[9] := FALSE;
   QW_STW[10] := FALSE;
   QW_STW[11] := FALSE;
   QW_STW[12] := FALSE;
   QW_STW[13] := FALSE;
   QW_STW[14] := FALSE;
   QW_STW[15] := FALSE;
   QW_HWValue := 19000;
   QDW_ScalledValue := 17.18027;
   QDW_Message[0] := FALSE;
   QDW_Message[1] := FALSE;
   QDW_Message[2] := FALSE;
   QDW_Message[3] := FALSE;
   QDW_Message[4] := FALSE;
   QDW_Message[5] := FALSE;
   QDW_Message[6] := FALSE;
   QDW_Message[7] := FALSE;
   QDW_Message[8] := FALSE;
   QDW_Message[9] := FALSE;
   QDW_Message[10] := FALSE;
   QDW_Message[11] := FALSE;
   QDW_Message[12] := FALSE;
   QDW_Message[13] := FALSE;
   QDW_Message[14] := TRUE;
   QDW_Message[15] := FALSE;
   QDW_Message[16] := FALSE;

END_DATA_BLOCK

DATA_BLOCK "AI_Tank2_DB"
{ S7_Optimized_Access := 'FALSE' }
AUTHOR : SimenCom
VERSION : 1.0
"Analog_In_UDT"

BEGIN

END_DATA_BLOCK

DATA_BLOCK "CalcVolume_Tank2_DB"
{ S7_Optimized_Access := 'FALSE' }
VERSION : 0.1
"CalculationVolume"

BEGIN
   IW_Radius := 1.468;
   IW_ValueFromSensor := 18.41001;
   IW_K_for_Tonnag := 1.35;
   IW_K_for_Level := 1.35;
   QW_Volume := 92.27883;
   QW_Tonnag := 124.5764;
   QW_RealLevel := 13.63704;
   sW_S := 6.766776;
   sW_Volume := 92.27883;
   sW_RealLevel := 13.63704;

END_DATA_BLOCK

DATA_BLOCK "UDT_AI_Tank2"
{ S7_Optimized_Access := 'FALSE' }
VERSION : 0.1
"UDT_Analog_In"

BEGIN
   IW_HW_UpLevel := 27648;
   IW_HW_LowLevel := 0;
   IDW_UpLevel := 25.0;
   IDW_LowLevel := 0.0;
   IDW_HiHi := 18.5;
   IDW_Hi := 18.0;
   IDW_Lo := 0.0;
   IDW_Lolo := 0.0;
   IW_DelayON_HiHi := 1;
   IW_DelayON_Hi := 1;
   IW_DelayON_Lo := 0;
   IW_DelayON_LoLo := 0;
   IDW_Simulation_Value := 0.0;
   IW_Time_Filter := 0;
   IW_CTW[0] := FALSE;
   IW_CTW[1] := FALSE;
   IW_CTW[2] := FALSE;
   IW_CTW[3] := FALSE;
   IW_CTW[4] := FALSE;
   IW_CTW[5] := FALSE;
   IW_CTW[6] := FALSE;
   IW_CTW[7] := FALSE;
   IW_CTW[8] := FALSE;
   IW_CTW[9] := FALSE;
   IW_CTW[10] := FALSE;
   IW_CTW[11] := FALSE;
   IW_CTW[12] := FALSE;
   IW_CTW[13] := FALSE;
   IW_CTW[14] := FALSE;
   IW_CTW[15] := FALSE;
   IDW_K_Mult := 1.0;
   IDW_DeadZone := 0.0;
   IBt_Enable_ControlLevel[0] := FALSE;
   IBt_Enable_ControlLevel[1] := FALSE;
   IBt_Enable_ControlLevel[2] := FALSE;
   IBt_Enable_ControlLevel[3] := FALSE;
   IBt_Enable_ControlLevel[4] := FALSE;
   IBt_Enable_ControlLevel[5] := FALSE;
   IBt_Enable_ControlLevel[6] := FALSE;
   IBt_Enable_ControlLevel[7] := FALSE;
   IBt_Block_ControlLevel[0] := FALSE;
   IBt_Block_ControlLevel[1] := FALSE;
   IBt_Block_ControlLevel[2] := FALSE;
   IBt_Block_ControlLevel[3] := FALSE;
   IBt_Block_ControlLevel[4] := FALSE;
   IBt_Block_ControlLevel[5] := FALSE;
   IBt_Block_ControlLevel[6] := FALSE;
   IBt_Block_ControlLevel[7] := FALSE;
   QW_STW[0] := FALSE;
   QW_STW[1] := FALSE;
   QW_STW[2] := TRUE;
   QW_STW[3] := FALSE;
   QW_STW[4] := FALSE;
   QW_STW[5] := FALSE;
   QW_STW[6] := FALSE;
   QW_STW[7] := FALSE;
   QW_STW[8] := FALSE;
   QW_STW[9] := FALSE;
   QW_STW[10] := FALSE;
   QW_STW[11] := FALSE;
   QW_STW[12] := FALSE;
   QW_STW[13] := FALSE;
   QW_STW[14] := FALSE;
   QW_STW[15] := FALSE;
   QW_HWValue := 20356;
   QDW_ScalledValue := 18.40639;
   QDW_Message[0] := FALSE;
   QDW_Message[1] := FALSE;
   QDW_Message[2] := FALSE;
   QDW_Message[3] := FALSE;
   QDW_Message[4] := FALSE;
   QDW_Message[5] := FALSE;
   QDW_Message[6] := FALSE;
   QDW_Message[7] := FALSE;
   QDW_Message[8] := FALSE;
   QDW_Message[9] := FALSE;
   QDW_Message[10] := FALSE;
   QDW_Message[11] := FALSE;
   QDW_Message[12] := FALSE;
   QDW_Message[13] := FALSE;
   QDW_Message[14] := FALSE;
   QDW_Message[15] := FALSE;
   QDW_Message[16] := FALSE;

END_DATA_BLOCK

DATA_BLOCK "AI_Tank3_DB"
{ S7_Optimized_Access := 'FALSE' }
AUTHOR : SimenCom
VERSION : 1.0
"Analog_In_UDT"

BEGIN

END_DATA_BLOCK

DATA_BLOCK "CalcVolume_Tank3_DB"
{ S7_Optimized_Access := 'FALSE' }
VERSION : 0.1
"CalculationVolume"

BEGIN
   IW_Radius := 1.468;
   IW_ValueFromSensor := 9.675202;
   IW_K_for_Tonnag := 1.35;
   IW_K_for_Level := 1.35;
   QW_Volume := 48.49624;
   QW_Tonnag := 65.46992;
   QW_RealLevel := 7.166816;
   sW_S := 6.766776;
   sW_Volume := 48.49624;
   sW_RealLevel := 7.166816;

END_DATA_BLOCK

DATA_BLOCK "UDT_AI_Tank3"
{ S7_Optimized_Access := 'FALSE' }
VERSION : 0.1
"UDT_Analog_In"

BEGIN
   IW_HW_UpLevel := 27648;
   IW_HW_LowLevel := 0;
   IDW_UpLevel := 25.0;
   IDW_LowLevel := 0.0;
   IDW_HiHi := 18.5;
   IDW_Hi := 18.0;
   IDW_Lo := 0.0;
   IDW_Lolo := 4.0;
   IW_DelayON_HiHi := 1;
   IW_DelayON_Hi := 1;
   IW_DelayON_Lo := 0;
   IW_DelayON_LoLo := 0;
   IDW_Simulation_Value := 0.0;
   IW_Time_Filter := 0;
   IW_CTW[0] := FALSE;
   IW_CTW[1] := FALSE;
   IW_CTW[2] := FALSE;
   IW_CTW[3] := FALSE;
   IW_CTW[4] := FALSE;
   IW_CTW[5] := FALSE;
   IW_CTW[6] := FALSE;
   IW_CTW[7] := FALSE;
   IW_CTW[8] := FALSE;
   IW_CTW[9] := FALSE;
   IW_CTW[10] := FALSE;
   IW_CTW[11] := FALSE;
   IW_CTW[12] := FALSE;
   IW_CTW[13] := FALSE;
   IW_CTW[14] := FALSE;
   IW_CTW[15] := FALSE;
   IDW_K_Mult := 1.0;
   IDW_DeadZone := 0.0;
   IBt_Enable_ControlLevel[0] := TRUE;
   IBt_Enable_ControlLevel[1] := TRUE;
   IBt_Enable_ControlLevel[2] := FALSE;
   IBt_Enable_ControlLevel[3] := FALSE;
   IBt_Enable_ControlLevel[4] := FALSE;
   IBt_Enable_ControlLevel[5] := FALSE;
   IBt_Enable_ControlLevel[6] := FALSE;
   IBt_Enable_ControlLevel[7] := FALSE;
   IBt_Block_ControlLevel[0] := FALSE;
   IBt_Block_ControlLevel[1] := FALSE;
   IBt_Block_ControlLevel[2] := FALSE;
   IBt_Block_ControlLevel[3] := FALSE;
   IBt_Block_ControlLevel[4] := FALSE;
   IBt_Block_ControlLevel[5] := FALSE;
   IBt_Block_ControlLevel[6] := FALSE;
   IBt_Block_ControlLevel[7] := FALSE;
   QW_STW[0] := FALSE;
   QW_STW[1] := FALSE;
   QW_STW[2] := TRUE;
   QW_STW[3] := FALSE;
   QW_STW[4] := FALSE;
   QW_STW[5] := FALSE;
   QW_STW[6] := FALSE;
   QW_STW[7] := FALSE;
   QW_STW[8] := FALSE;
   QW_STW[9] := FALSE;
   QW_STW[10] := FALSE;
   QW_STW[11] := FALSE;
   QW_STW[12] := FALSE;
   QW_STW[13] := FALSE;
   QW_STW[14] := FALSE;
   QW_STW[15] := FALSE;
   QW_HWValue := 10704;
   QDW_ScalledValue := 9.67882;
   QDW_Message[0] := FALSE;
   QDW_Message[1] := FALSE;
   QDW_Message[2] := FALSE;
   QDW_Message[3] := FALSE;
   QDW_Message[4] := FALSE;
   QDW_Message[5] := FALSE;
   QDW_Message[6] := FALSE;
   QDW_Message[7] := FALSE;
   QDW_Message[8] := FALSE;
   QDW_Message[9] := FALSE;
   QDW_Message[10] := FALSE;
   QDW_Message[11] := FALSE;
   QDW_Message[12] := FALSE;
   QDW_Message[13] := FALSE;
   QDW_Message[14] := FALSE;
   QDW_Message[15] := FALSE;
   QDW_Message[16] := FALSE;

END_DATA_BLOCK

DATA_BLOCK "AI_Tank4_DB"
{ S7_Optimized_Access := 'FALSE' }
AUTHOR : SimenCom
VERSION : 1.0
"Analog_In_UDT"

BEGIN

END_DATA_BLOCK

DATA_BLOCK "CalcVolume_Tank4_DB"
{ S7_Optimized_Access := 'FALSE' }
VERSION : 0.1
"CalculationVolume"

BEGIN
   IW_Radius := 1.468;
   IW_ValueFromSensor := 13.19083;
   IW_K_for_Tonnag := 1.35;
   IW_K_for_Level := 1.35;
   QW_Volume := 66.11805;
   QW_Tonnag := 89.25937;
   QW_RealLevel := 9.770983;
   sW_S := 6.766776;
   sW_Volume := 66.11805;
   sW_RealLevel := 9.770983;

END_DATA_BLOCK

DATA_BLOCK "UDT_AI_Tank4"
{ S7_Optimized_Access := 'FALSE' }
VERSION : 0.1
"UDT_Analog_In"

BEGIN
   IW_HW_UpLevel := 27648;
   IW_HW_LowLevel := 0;
   IDW_UpLevel := 25.0;
   IDW_LowLevel := 0.0;
   IDW_HiHi := 18.5;
   IDW_Hi := 18.0;
   IDW_Lo := 0.0;
   IDW_Lolo := 0.0;
   IW_DelayON_HiHi := 1;
   IW_DelayON_Hi := 1;
   IW_DelayON_Lo := 0;
   IW_DelayON_LoLo := 0;
   IDW_Simulation_Value := 0.0;
   IW_Time_Filter := 0;
   IW_CTW[0] := FALSE;
   IW_CTW[1] := FALSE;
   IW_CTW[2] := FALSE;
   IW_CTW[3] := FALSE;
   IW_CTW[4] := FALSE;
   IW_CTW[5] := FALSE;
   IW_CTW[6] := FALSE;
   IW_CTW[7] := FALSE;
   IW_CTW[8] := FALSE;
   IW_CTW[9] := FALSE;
   IW_CTW[10] := FALSE;
   IW_CTW[11] := FALSE;
   IW_CTW[12] := FALSE;
   IW_CTW[13] := FALSE;
   IW_CTW[14] := FALSE;
   IW_CTW[15] := FALSE;
   IDW_K_Mult := 1.0;
   IDW_DeadZone := 0.0;
   IBt_Enable_ControlLevel[0] := TRUE;
   IBt_Enable_ControlLevel[1] := TRUE;
   IBt_Enable_ControlLevel[2] := FALSE;
   IBt_Enable_ControlLevel[3] := FALSE;
   IBt_Enable_ControlLevel[4] := FALSE;
   IBt_Enable_ControlLevel[5] := FALSE;
   IBt_Enable_ControlLevel[6] := FALSE;
   IBt_Enable_ControlLevel[7] := FALSE;
   IBt_Block_ControlLevel[0] := FALSE;
   IBt_Block_ControlLevel[1] := FALSE;
   IBt_Block_ControlLevel[2] := FALSE;
   IBt_Block_ControlLevel[3] := FALSE;
   IBt_Block_ControlLevel[4] := FALSE;
   IBt_Block_ControlLevel[5] := FALSE;
   IBt_Block_ControlLevel[6] := FALSE;
   IBt_Block_ControlLevel[7] := FALSE;
   QW_STW[0] := FALSE;
   QW_STW[1] := FALSE;
   QW_STW[2] := TRUE;
   QW_STW[3] := FALSE;
   QW_STW[4] := FALSE;
   QW_STW[5] := FALSE;
   QW_STW[6] := FALSE;
   QW_STW[7] := FALSE;
   QW_STW[8] := FALSE;
   QW_STW[9] := FALSE;
   QW_STW[10] := FALSE;
   QW_STW[11] := FALSE;
   QW_STW[12] := FALSE;
   QW_STW[13] := FALSE;
   QW_STW[14] := FALSE;
   QW_STW[15] := FALSE;
   QW_HWValue := 14588;
   QDW_ScalledValue := 13.19083;
   QDW_Message[0] := FALSE;
   QDW_Message[1] := FALSE;
   QDW_Message[2] := FALSE;
   QDW_Message[3] := FALSE;
   QDW_Message[4] := FALSE;
   QDW_Message[5] := FALSE;
   QDW_Message[6] := FALSE;
   QDW_Message[7] := FALSE;
   QDW_Message[8] := FALSE;
   QDW_Message[9] := FALSE;
   QDW_Message[10] := FALSE;
   QDW_Message[11] := FALSE;
   QDW_Message[12] := FALSE;
   QDW_Message[13] := FALSE;
   QDW_Message[14] := FALSE;
   QDW_Message[15] := FALSE;
   QDW_Message[16] := FALSE;

END_DATA_BLOCK

DATA_BLOCK "AI_Tank5_DB"
{ S7_Optimized_Access := 'FALSE' }
AUTHOR : SimenCom
VERSION : 1.0
"Analog_In_UDT"

BEGIN

END_DATA_BLOCK

DATA_BLOCK "CalcVolume_Tank5_DB"
{ S7_Optimized_Access := 'FALSE' }
VERSION : 0.1
"CalculationVolume"

BEGIN
   IW_Radius := 1.468;
   IW_ValueFromSensor := 18.26172;
   IW_K_for_Tonnag := 1.35;
   IW_K_for_Level := 1.35;
   QW_Volume := 91.53552;
   QW_Tonnag := 123.573;
   QW_RealLevel := 13.5272;
   sW_S := 6.766776;
   sW_Volume := 91.53552;
   sW_RealLevel := 13.5272;

END_DATA_BLOCK

DATA_BLOCK "UDT_AI_Tank5"
{ S7_Optimized_Access := 'FALSE' }
VERSION : 0.1
"UDT_Analog_In"

BEGIN
   IW_HW_UpLevel := 27648;
   IW_HW_LowLevel := 0;
   IDW_UpLevel := 25.0;
   IDW_LowLevel := 0.0;
   IDW_HiHi := 18.5;
   IDW_Hi := 18.0;
   IDW_Lo := 0.0;
   IDW_Lolo := 0.0;
   IW_DelayON_HiHi := 1;
   IW_DelayON_Hi := 1;
   IW_DelayON_Lo := 0;
   IW_DelayON_LoLo := 0;
   IDW_Simulation_Value := 0.0;
   IW_Time_Filter := 0;
   IW_CTW[0] := FALSE;
   IW_CTW[1] := FALSE;
   IW_CTW[2] := FALSE;
   IW_CTW[3] := FALSE;
   IW_CTW[4] := FALSE;
   IW_CTW[5] := FALSE;
   IW_CTW[6] := FALSE;
   IW_CTW[7] := FALSE;
   IW_CTW[8] := FALSE;
   IW_CTW[9] := FALSE;
   IW_CTW[10] := FALSE;
   IW_CTW[11] := FALSE;
   IW_CTW[12] := FALSE;
   IW_CTW[13] := FALSE;
   IW_CTW[14] := FALSE;
   IW_CTW[15] := FALSE;
   IDW_K_Mult := 1.0;
   IDW_DeadZone := 0.0;
   IBt_Enable_ControlLevel[0] := TRUE;
   IBt_Enable_ControlLevel[1] := TRUE;
   IBt_Enable_ControlLevel[2] := FALSE;
   IBt_Enable_ControlLevel[3] := FALSE;
   IBt_Enable_ControlLevel[4] := FALSE;
   IBt_Enable_ControlLevel[5] := FALSE;
   IBt_Enable_ControlLevel[6] := FALSE;
   IBt_Enable_ControlLevel[7] := FALSE;
   IBt_Block_ControlLevel[0] := FALSE;
   IBt_Block_ControlLevel[1] := FALSE;
   IBt_Block_ControlLevel[2] := FALSE;
   IBt_Block_ControlLevel[3] := FALSE;
   IBt_Block_ControlLevel[4] := FALSE;
   IBt_Block_ControlLevel[5] := FALSE;
   IBt_Block_ControlLevel[6] := FALSE;
   IBt_Block_ControlLevel[7] := FALSE;
   QW_STW[0] := FALSE;
   QW_STW[1] := TRUE;
   QW_STW[2] := FALSE;
   QW_STW[3] := FALSE;
   QW_STW[4] := FALSE;
   QW_STW[5] := TRUE;
   QW_STW[6] := FALSE;
   QW_STW[7] := FALSE;
   QW_STW[8] := FALSE;
   QW_STW[9] := FALSE;
   QW_STW[10] := FALSE;
   QW_STW[11] := FALSE;
   QW_STW[12] := FALSE;
   QW_STW[13] := FALSE;
   QW_STW[14] := FALSE;
   QW_STW[15] := FALSE;
   QW_HWValue := 20196;
   QDW_ScalledValue := 18.26172;
   QDW_Message[0] := FALSE;
   QDW_Message[1] := FALSE;
   QDW_Message[2] := FALSE;
   QDW_Message[3] := FALSE;
   QDW_Message[4] := FALSE;
   QDW_Message[5] := FALSE;
   QDW_Message[6] := FALSE;
   QDW_Message[7] := FALSE;
   QDW_Message[8] := FALSE;
   QDW_Message[9] := FALSE;
   QDW_Message[10] := FALSE;
   QDW_Message[11] := FALSE;
   QDW_Message[12] := FALSE;
   QDW_Message[13] := FALSE;
   QDW_Message[14] := TRUE;
   QDW_Message[15] := FALSE;
   QDW_Message[16] := FALSE;

END_DATA_BLOCK

DATA_BLOCK "AI_Tank6_DB"
{ S7_Optimized_Access := 'FALSE' }
AUTHOR : SimenCom
VERSION : 1.0
"Analog_In_UDT"

BEGIN

END_DATA_BLOCK

DATA_BLOCK "CalcVolume_Tank6_DB"
{ S7_Optimized_Access := 'FALSE' }
VERSION : 0.1
"CalculationVolume"

BEGIN
   IW_Radius := 1.468;
   IW_ValueFromSensor := 18.24364;
   IW_K_for_Tonnag := 1.35;
   IW_K_for_Level := 1.35;
   QW_Volume := 91.44489;
   QW_Tonnag := 123.4506;
   QW_RealLevel := 13.5138;
   sW_S := 6.766776;
   sW_Volume := 91.44489;
   sW_RealLevel := 13.5138;

END_DATA_BLOCK

DATA_BLOCK "UDT_AI_Tank6"
{ S7_Optimized_Access := 'FALSE' }
VERSION : 0.1
"UDT_Analog_In"

BEGIN
   IW_HW_UpLevel := 27648;
   IW_HW_LowLevel := 0;
   IDW_UpLevel := 25.0;
   IDW_LowLevel := 0.0;
   IDW_HiHi := 18.5;
   IDW_Hi := 18.0;
   IDW_Lo := 0.0;
   IDW_Lolo := 0.0;
   IW_DelayON_HiHi := 1;
   IW_DelayON_Hi := 1;
   IW_DelayON_Lo := 0;
   IW_DelayON_LoLo := 0;
   IDW_Simulation_Value := 0.0;
   IW_Time_Filter := 0;
   IW_CTW[0] := FALSE;
   IW_CTW[1] := FALSE;
   IW_CTW[2] := FALSE;
   IW_CTW[3] := FALSE;
   IW_CTW[4] := FALSE;
   IW_CTW[5] := FALSE;
   IW_CTW[6] := FALSE;
   IW_CTW[7] := FALSE;
   IW_CTW[8] := FALSE;
   IW_CTW[9] := FALSE;
   IW_CTW[10] := FALSE;
   IW_CTW[11] := FALSE;
   IW_CTW[12] := FALSE;
   IW_CTW[13] := FALSE;
   IW_CTW[14] := FALSE;
   IW_CTW[15] := FALSE;
   IDW_K_Mult := 1.0;
   IDW_DeadZone := 0.0;
   IBt_Enable_ControlLevel[0] := TRUE;
   IBt_Enable_ControlLevel[1] := TRUE;
   IBt_Enable_ControlLevel[2] := FALSE;
   IBt_Enable_ControlLevel[3] := FALSE;
   IBt_Enable_ControlLevel[4] := FALSE;
   IBt_Enable_ControlLevel[5] := FALSE;
   IBt_Enable_ControlLevel[6] := FALSE;
   IBt_Enable_ControlLevel[7] := FALSE;
   IBt_Block_ControlLevel[0] := FALSE;
   IBt_Block_ControlLevel[1] := FALSE;
   IBt_Block_ControlLevel[2] := FALSE;
   IBt_Block_ControlLevel[3] := FALSE;
   IBt_Block_ControlLevel[4] := FALSE;
   IBt_Block_ControlLevel[5] := FALSE;
   IBt_Block_ControlLevel[6] := FALSE;
   IBt_Block_ControlLevel[7] := FALSE;
   QW_STW[0] := FALSE;
   QW_STW[1] := TRUE;
   QW_STW[2] := FALSE;
   QW_STW[3] := FALSE;
   QW_STW[4] := FALSE;
   QW_STW[5] := TRUE;
   QW_STW[6] := FALSE;
   QW_STW[7] := FALSE;
   QW_STW[8] := FALSE;
   QW_STW[9] := FALSE;
   QW_STW[10] := FALSE;
   QW_STW[11] := FALSE;
   QW_STW[12] := FALSE;
   QW_STW[13] := FALSE;
   QW_STW[14] := FALSE;
   QW_STW[15] := FALSE;
   QW_HWValue := 20172;
   QDW_ScalledValue := 18.24002;
   QDW_Message[0] := FALSE;
   QDW_Message[1] := FALSE;
   QDW_Message[2] := FALSE;
   QDW_Message[3] := FALSE;
   QDW_Message[4] := FALSE;
   QDW_Message[5] := FALSE;
   QDW_Message[6] := FALSE;
   QDW_Message[7] := FALSE;
   QDW_Message[8] := FALSE;
   QDW_Message[9] := FALSE;
   QDW_Message[10] := FALSE;
   QDW_Message[11] := FALSE;
   QDW_Message[12] := FALSE;
   QDW_Message[13] := FALSE;
   QDW_Message[14] := TRUE;
   QDW_Message[15] := FALSE;
   QDW_Message[16] := FALSE;

END_DATA_BLOCK

DATA_BLOCK "AI_Tank7_DB"
{ S7_Optimized_Access := 'FALSE' }
AUTHOR : SimenCom
VERSION : 1.0
"Analog_In_UDT"

BEGIN

END_DATA_BLOCK

DATA_BLOCK "CalcVolume_Tank7_DB"
{ S7_Optimized_Access := 'FALSE' }
VERSION : 0.1
"CalculationVolume"

BEGIN
   IW_Radius := 1.468;
   IW_ValueFromSensor := 13.7406;
   IW_K_for_Tonnag := 1.35;
   IW_K_for_Level := 1.35;
   QW_Volume := 68.87373;
   QW_Tonnag := 92.97953;
   QW_RealLevel := 10.17822;
   sW_S := 6.766776;
   sW_Volume := 68.87373;
   sW_RealLevel := 10.17822;

END_DATA_BLOCK

DATA_BLOCK "UDT_AI_Tank7"
{ S7_Optimized_Access := 'FALSE' }
VERSION : 0.1
"UDT_Analog_In"

BEGIN
   IW_HW_UpLevel := 27648;
   IW_HW_LowLevel := 0;
   IDW_UpLevel := 25.0;
   IDW_LowLevel := 0.0;
   IDW_HiHi := 18.5;
   IDW_Hi := 18.0;
   IDW_Lo := 0.0;
   IDW_Lolo := 0.0;
   IW_DelayON_HiHi := 1;
   IW_DelayON_Hi := 1;
   IW_DelayON_Lo := 0;
   IW_DelayON_LoLo := 0;
   IDW_Simulation_Value := 0.0;
   IW_Time_Filter := 0;
   IW_CTW[0] := FALSE;
   IW_CTW[1] := FALSE;
   IW_CTW[2] := FALSE;
   IW_CTW[3] := FALSE;
   IW_CTW[4] := FALSE;
   IW_CTW[5] := FALSE;
   IW_CTW[6] := FALSE;
   IW_CTW[7] := FALSE;
   IW_CTW[8] := FALSE;
   IW_CTW[9] := FALSE;
   IW_CTW[10] := FALSE;
   IW_CTW[11] := FALSE;
   IW_CTW[12] := FALSE;
   IW_CTW[13] := FALSE;
   IW_CTW[14] := FALSE;
   IW_CTW[15] := FALSE;
   IDW_K_Mult := 1.0;
   IDW_DeadZone := 0.0;
   IBt_Enable_ControlLevel[0] := TRUE;
   IBt_Enable_ControlLevel[1] := TRUE;
   IBt_Enable_ControlLevel[2] := FALSE;
   IBt_Enable_ControlLevel[3] := FALSE;
   IBt_Enable_ControlLevel[4] := FALSE;
   IBt_Enable_ControlLevel[5] := FALSE;
   IBt_Enable_ControlLevel[6] := FALSE;
   IBt_Enable_ControlLevel[7] := FALSE;
   IBt_Block_ControlLevel[0] := FALSE;
   IBt_Block_ControlLevel[1] := FALSE;
   IBt_Block_ControlLevel[2] := FALSE;
   IBt_Block_ControlLevel[3] := FALSE;
   IBt_Block_ControlLevel[4] := FALSE;
   IBt_Block_ControlLevel[5] := FALSE;
   IBt_Block_ControlLevel[6] := FALSE;
   IBt_Block_ControlLevel[7] := FALSE;
   QW_STW[0] := FALSE;
   QW_STW[1] := FALSE;
   QW_STW[2] := TRUE;
   QW_STW[3] := FALSE;
   QW_STW[4] := FALSE;
   QW_STW[5] := FALSE;
   QW_STW[6] := FALSE;
   QW_STW[7] := FALSE;
   QW_STW[8] := FALSE;
   QW_STW[9] := FALSE;
   QW_STW[10] := FALSE;
   QW_STW[11] := FALSE;
   QW_STW[12] := FALSE;
   QW_STW[13] := FALSE;
   QW_STW[14] := FALSE;
   QW_STW[15] := FALSE;
   QW_HWValue := 15200;
   QDW_ScalledValue := 13.74421;
   QDW_Message[0] := FALSE;
   QDW_Message[1] := FALSE;
   QDW_Message[2] := FALSE;
   QDW_Message[3] := FALSE;
   QDW_Message[4] := FALSE;
   QDW_Message[5] := FALSE;
   QDW_Message[6] := FALSE;
   QDW_Message[7] := FALSE;
   QDW_Message[8] := FALSE;
   QDW_Message[9] := FALSE;
   QDW_Message[10] := FALSE;
   QDW_Message[11] := FALSE;
   QDW_Message[12] := FALSE;
   QDW_Message[13] := FALSE;
   QDW_Message[14] := FALSE;
   QDW_Message[15] := FALSE;
   QDW_Message[16] := FALSE;

END_DATA_BLOCK

DATA_BLOCK "AI_Tank8_DB"
{ S7_Optimized_Access := 'FALSE' }
AUTHOR : SimenCom
VERSION : 1.0
"Analog_In_UDT"

BEGIN

END_DATA_BLOCK

DATA_BLOCK "CalcVolume_Tank8_DB"
{ S7_Optimized_Access := 'FALSE' }
VERSION : 0.1
"CalculationVolume"

BEGIN
   IW_Radius := 1.468;
   IW_ValueFromSensor := 18.48597;
   IW_K_for_Tonnag := 1.35;
   IW_K_for_Level := 1.35;
   QW_Volume := 92.65955;
   QW_Tonnag := 125.0904;
   QW_RealLevel := 13.69331;
   sW_S := 6.766776;
   sW_Volume := 92.65955;
   sW_RealLevel := 13.69331;

END_DATA_BLOCK

DATA_BLOCK "UDT_AI_Tank8"
{ S7_Optimized_Access := 'FALSE' }
VERSION : 0.1
"UDT_Analog_In"

BEGIN
   IW_HW_UpLevel := 27648;
   IW_HW_LowLevel := 0;
   IDW_UpLevel := 25.0;
   IDW_LowLevel := 0.0;
   IDW_HiHi := 18.5;
   IDW_Hi := 18.0;
   IDW_Lo := 0.0;
   IDW_Lolo := 0.0;
   IW_DelayON_HiHi := 1;
   IW_DelayON_Hi := 1;
   IW_DelayON_Lo := 0;
   IW_DelayON_LoLo := 0;
   IDW_Simulation_Value := 0.0;
   IW_Time_Filter := 0;
   IW_CTW[0] := FALSE;
   IW_CTW[1] := FALSE;
   IW_CTW[2] := FALSE;
   IW_CTW[3] := FALSE;
   IW_CTW[4] := FALSE;
   IW_CTW[5] := FALSE;
   IW_CTW[6] := FALSE;
   IW_CTW[7] := FALSE;
   IW_CTW[8] := FALSE;
   IW_CTW[9] := FALSE;
   IW_CTW[10] := FALSE;
   IW_CTW[11] := FALSE;
   IW_CTW[12] := FALSE;
   IW_CTW[13] := FALSE;
   IW_CTW[14] := FALSE;
   IW_CTW[15] := FALSE;
   IDW_K_Mult := 1.0;
   IDW_DeadZone := 0.0;
   IBt_Enable_ControlLevel[0] := TRUE;
   IBt_Enable_ControlLevel[1] := TRUE;
   IBt_Enable_ControlLevel[2] := FALSE;
   IBt_Enable_ControlLevel[3] := FALSE;
   IBt_Enable_ControlLevel[4] := FALSE;
   IBt_Enable_ControlLevel[5] := FALSE;
   IBt_Enable_ControlLevel[6] := FALSE;
   IBt_Enable_ControlLevel[7] := FALSE;
   IBt_Block_ControlLevel[0] := FALSE;
   IBt_Block_ControlLevel[1] := FALSE;
   IBt_Block_ControlLevel[2] := FALSE;
   IBt_Block_ControlLevel[3] := FALSE;
   IBt_Block_ControlLevel[4] := FALSE;
   IBt_Block_ControlLevel[5] := FALSE;
   IBt_Block_ControlLevel[6] := FALSE;
   IBt_Block_ControlLevel[7] := FALSE;
   QW_STW[0] := FALSE;
   QW_STW[1] := TRUE;
   QW_STW[2] := FALSE;
   QW_STW[3] := FALSE;
   QW_STW[4] := FALSE;
   QW_STW[5] := TRUE;
   QW_STW[6] := FALSE;
   QW_STW[7] := FALSE;
   QW_STW[8] := FALSE;
   QW_STW[9] := FALSE;
   QW_STW[10] := FALSE;
   QW_STW[11] := FALSE;
   QW_STW[12] := FALSE;
   QW_STW[13] := FALSE;
   QW_STW[14] := FALSE;
   QW_STW[15] := FALSE;
   QW_HWValue := 20444;
   QDW_ScalledValue := 18.48597;
   QDW_Message[0] := FALSE;
   QDW_Message[1] := FALSE;
   QDW_Message[2] := FALSE;
   QDW_Message[3] := FALSE;
   QDW_Message[4] := FALSE;
   QDW_Message[5] := FALSE;
   QDW_Message[6] := FALSE;
   QDW_Message[7] := FALSE;
   QDW_Message[8] := FALSE;
   QDW_Message[9] := FALSE;
   QDW_Message[10] := FALSE;
   QDW_Message[11] := FALSE;
   QDW_Message[12] := FALSE;
   QDW_Message[13] := FALSE;
   QDW_Message[14] := TRUE;
   QDW_Message[15] := FALSE;
   QDW_Message[16] := FALSE;

END_DATA_BLOCK

DATA_BLOCK "AI_Tank9_DB"
{ S7_Optimized_Access := 'FALSE' }
AUTHOR : SimenCom
VERSION : 1.0
"Analog_In_UDT"

BEGIN

END_DATA_BLOCK

DATA_BLOCK "CalcVolume_Tank9_DB"
{ S7_Optimized_Access := 'FALSE' }
VERSION : 0.1
"CalculationVolume"

BEGIN
   IW_Radius := 1.468;
   IW_ValueFromSensor := 18.20747;
   IW_K_for_Tonnag := 1.35;
   IW_K_for_Level := 1.35;
   QW_Volume := 91.26359;
   QW_Tonnag := 123.2058;
   QW_RealLevel := 13.48701;
   sW_S := 6.766776;
   sW_Volume := 91.26359;
   sW_RealLevel := 13.48701;

END_DATA_BLOCK

DATA_BLOCK "UDT_AI_Tank9"
{ S7_Optimized_Access := 'FALSE' }
VERSION : 0.1
"UDT_Analog_In"

BEGIN
   IW_HW_UpLevel := 27648;
   IW_HW_LowLevel := 0;
   IDW_UpLevel := 25.0;
   IDW_LowLevel := 0.0;
   IDW_HiHi := 18.5;
   IDW_Hi := 18.0;
   IDW_Lo := 0.0;
   IDW_Lolo := 0.0;
   IW_DelayON_HiHi := 1;
   IW_DelayON_Hi := 1;
   IW_DelayON_Lo := 0;
   IW_DelayON_LoLo := 0;
   IDW_Simulation_Value := 0.0;
   IW_Time_Filter := 0;
   IW_CTW[0] := FALSE;
   IW_CTW[1] := FALSE;
   IW_CTW[2] := FALSE;
   IW_CTW[3] := FALSE;
   IW_CTW[4] := FALSE;
   IW_CTW[5] := FALSE;
   IW_CTW[6] := FALSE;
   IW_CTW[7] := FALSE;
   IW_CTW[8] := FALSE;
   IW_CTW[9] := FALSE;
   IW_CTW[10] := FALSE;
   IW_CTW[11] := FALSE;
   IW_CTW[12] := FALSE;
   IW_CTW[13] := FALSE;
   IW_CTW[14] := FALSE;
   IW_CTW[15] := FALSE;
   IDW_K_Mult := 1.0;
   IDW_DeadZone := 0.0;
   IBt_Enable_ControlLevel[0] := TRUE;
   IBt_Enable_ControlLevel[1] := TRUE;
   IBt_Enable_ControlLevel[2] := FALSE;
   IBt_Enable_ControlLevel[3] := FALSE;
   IBt_Enable_ControlLevel[4] := FALSE;
   IBt_Enable_ControlLevel[5] := FALSE;
   IBt_Enable_ControlLevel[6] := FALSE;
   IBt_Enable_ControlLevel[7] := FALSE;
   IBt_Block_ControlLevel[0] := FALSE;
   IBt_Block_ControlLevel[1] := FALSE;
   IBt_Block_ControlLevel[2] := FALSE;
   IBt_Block_ControlLevel[3] := FALSE;
   IBt_Block_ControlLevel[4] := FALSE;
   IBt_Block_ControlLevel[5] := FALSE;
   IBt_Block_ControlLevel[6] := FALSE;
   IBt_Block_ControlLevel[7] := FALSE;
   QW_STW[0] := FALSE;
   QW_STW[1] := TRUE;
   QW_STW[2] := FALSE;
   QW_STW[3] := FALSE;
   QW_STW[4] := FALSE;
   QW_STW[5] := TRUE;
   QW_STW[6] := FALSE;
   QW_STW[7] := FALSE;
   QW_STW[8] := FALSE;
   QW_STW[9] := FALSE;
   QW_STW[10] := FALSE;
   QW_STW[11] := FALSE;
   QW_STW[12] := FALSE;
   QW_STW[13] := FALSE;
   QW_STW[14] := FALSE;
   QW_STW[15] := FALSE;
   QW_HWValue := 20136;
   QDW_ScalledValue := 18.20747;
   QDW_Message[0] := FALSE;
   QDW_Message[1] := FALSE;
   QDW_Message[2] := FALSE;
   QDW_Message[3] := FALSE;
   QDW_Message[4] := FALSE;
   QDW_Message[5] := FALSE;
   QDW_Message[6] := FALSE;
   QDW_Message[7] := FALSE;
   QDW_Message[8] := FALSE;
   QDW_Message[9] := FALSE;
   QDW_Message[10] := FALSE;
   QDW_Message[11] := FALSE;
   QDW_Message[12] := FALSE;
   QDW_Message[13] := FALSE;
   QDW_Message[14] := TRUE;
   QDW_Message[15] := FALSE;
   QDW_Message[16] := FALSE;

END_DATA_BLOCK

ORGANIZATION_BLOCK "Main"   // OB1, FBD, ProgramCycle
TITLE = "Main Program Sweep (Cycle)"
VERSION : 0.1
// stored: IsIECCheckEnabled false
   VAR_TEMP
      OB1_EV_CLASS : Byte;   // Bits 0-3 = 1 (Coming event), Bits 4-7 = 1 (Event class 1)
      OB1_SCAN_1 : Byte;   // 1 (Cold restart scan 1 of OB 1), 3 (Scan 2-n of OB 1)
      OB1_PRIORITY : Byte;   // Priority of OB Execution
      OB1_OB_NUMBR : Byte;   // 1 (Organization block 1, OB1)
      OB1_RESERVED_1 : Byte;   // Reserved for system
      OB1_RESERVED_2 : Byte;   // Reserved for system
      OB1_PREV_CYCLE : Int;   // Cycle time of previous OB1 scan (milliseconds)
      OB1_MIN_CYCLE : Int;   // Minimum cycle time of OB1 (milliseconds)
      OB1_MAX_CYCLE : Int;   // Maximum cycle time of OB1 (milliseconds)
      OB1_DATE_TIME : Date_And_Time;   // Date and time OB1 started
   END_VAR
BEGIN

REGION Network 1
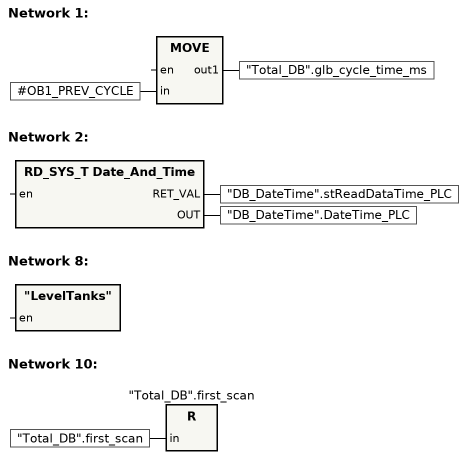
   "Total_DB".glb_cycle_time_ms := #OB1_PREV_CYCLE;
END_REGION

REGION Network 2
   "DB_DateTime".stReadDataTime_PLC := RD_SYS_T(OUT => "DB_DateTime".DateTime_PLC);
END_REGION

REGION Network 8
   "LevelTanks"();
END_REGION

REGION Network 10
   IF "Total_DB".first_scan THEN "Total_DB".first_scan := FALSE; END_IF;
END_REGION
END_ORGANIZATION_BLOCK

FUNCTION "LevelTanks" : Void
{ S7_Optimized_Access := 'FALSE' }
VERSION : 0.1

BEGIN
	
	REGION Polska - Tank 1
	    
	    "AI_Tank1_DB"(IB_Reset_PLC := "Total_DB".Restart_PLC,
	                  IB_Total_Reset := "Total_DB".Total_Reset_HMI,
	                  IB_EnablePowerControl := FALSE,
	                  IW_HW_UpLevel := 27648,
	                  IW_HW_LowLevel := 0,
	                  IW_Signal_from_Sensor := "Pol_sklad_sens",
	                  IUDT_Analog_In := "UDT_AI_Tank1");
	    
	 "CalcVolume_Tank1_DB"(IW_ValueFromSensor:="AI_Tank1_DB".QDW_ScalledValue);
	 
	END_REGION
	
	REGION Polska - Tank 2
	    
	    "AI_Tank2_DB"(IB_Reset_PLC := "Total_DB".Restart_PLC,
	                  IB_Total_Reset := "Total_DB".Total_Reset_HMI,
	                  IB_EnablePowerControl := FALSE,
	                  IW_HW_UpLevel := 27648,
	                  IW_HW_LowLevel := 0,
	                  IW_Signal_from_Sensor := "Pol_sens",
	                  IUDT_Analog_In := "UDT_AI_Tank2");
	    
	    "CalcVolume_Tank2_DB"(IW_ValueFromSensor := "AI_Tank2_DB".QDW_ScalledValue);
	    
	END_REGION
	
	REGION Polska - Tank 3
	    
	    "AI_Tank3_DB"(IB_Reset_PLC := "Total_DB".Restart_PLC,
	                  IB_Total_Reset := "Total_DB".Total_Reset_HMI,
	                  IB_EnablePowerControl := FALSE,
	                  IW_HW_UpLevel := 27648,
	                  IW_HW_LowLevel := 0,
	                  IW_Signal_from_Sensor := "IW_Tank3",
	                  IUDT_Analog_In := "UDT_AI_Tank3");
	    
	    "CalcVolume_Tank3_DB"(IW_ValueFromSensor := "AI_Tank3_DB".QDW_ScalledValue);
	    
	END_REGION
	
	REGION Polska - Tank 4
	    
	    "AI_Tank4_DB"(IB_Reset_PLC := "Total_DB".Restart_PLC,
	                  IB_Total_Reset := "Total_DB".Total_Reset_HMI,
	                  IB_EnablePowerControl := FALSE,
	                  IW_HW_UpLevel := 27648,
	                  IW_HW_LowLevel := 0,
	                  IW_Signal_from_Sensor := "IW_Tank4",
	                  IUDT_Analog_In := "UDT_AI_Tank4");
	    
	    "CalcVolume_Tank4_DB"(IW_ValueFromSensor := "AI_Tank4_DB".QDW_ScalledValue);
	    
	END_REGION
	
	REGION Polska - Tank 5
	    
	    "AI_Tank5_DB"(IB_Reset_PLC := "Total_DB".Restart_PLC,
	                  IB_Total_Reset := "Total_DB".Total_Reset_HMI,
	                  IB_EnablePowerControl := FALSE,
	                  IW_HW_UpLevel := 27648,
	                  IW_HW_LowLevel := 0,
	                  IW_Signal_from_Sensor := "IW_Tank5",
	                  IUDT_Analog_In := "UDT_AI_Tank5");
	    
	    "CalcVolume_Tank5_DB"(IW_ValueFromSensor := "AI_Tank5_DB".QDW_ScalledValue);
	    
	END_REGION
	
	REGION Polska - Tank 6
	    
	    "AI_Tank6_DB"(IB_Reset_PLC := "Total_DB".Restart_PLC,
	                  IB_Total_Reset := "Total_DB".Total_Reset_HMI,
	                  IB_EnablePowerControl := FALSE,
	                  IW_HW_UpLevel := 27648,
	                  IW_HW_LowLevel := 0,
	                  IW_Signal_from_Sensor := "IW_Tank6",
	                  IUDT_Analog_In := "UDT_AI_Tank6");
	    
	    "CalcVolume_Tank6_DB"(IW_ValueFromSensor := "AI_Tank6_DB".QDW_ScalledValue);
	    
	END_REGION
	
	REGION Polska - Tank 7
	    
	    "AI_Tank7_DB"(IB_Reset_PLC := "Total_DB".Restart_PLC,
	                  IB_Total_Reset := "Total_DB".Total_Reset_HMI,
	                  IB_EnablePowerControl := FALSE,
	                  IW_HW_UpLevel := 27648,
	                  IW_HW_LowLevel := 0,
	                  IW_Signal_from_Sensor := "IW_Tank7",
	                  IUDT_Analog_In := "UDT_AI_Tank7");
	    
	    "CalcVolume_Tank7_DB"(IW_ValueFromSensor := "AI_Tank7_DB".QDW_ScalledValue);
	    
	END_REGION
	
	REGION Polska - Tank 8
	    
	    "AI_Tank8_DB"(IB_Reset_PLC := "Total_DB".Restart_PLC,
	                  IB_Total_Reset := "Total_DB".Total_Reset_HMI,
	                  IB_EnablePowerControl := FALSE,
	                  IW_HW_UpLevel := 27648,
	                  IW_HW_LowLevel := 0,
	                  IW_Signal_from_Sensor := "IW_Tank8",
	                  IUDT_Analog_In := "UDT_AI_Tank8");
	    
	    "CalcVolume_Tank8_DB"(IW_ValueFromSensor := "AI_Tank8_DB".QDW_ScalledValue);
	    
	END_REGION
	
	REGION Polska - Tank 9
	    
	    "AI_Tank9_DB"(IB_Reset_PLC := "Total_DB".Restart_PLC,
	                  IB_Total_Reset := "Total_DB".Total_Reset_HMI,
	                  IB_EnablePowerControl := FALSE,
	                  IW_HW_UpLevel := 27648,
	                  IW_HW_LowLevel := 0,
	                  IW_Signal_from_Sensor := "IW_Tank9",
	                  IUDT_Analog_In := "UDT_AI_Tank9");
	    
	    "CalcVolume_Tank9_DB"(IW_ValueFromSensor := "AI_Tank9_DB".QDW_ScalledValue);
	    
	END_REGION
	
	REGION Polska - Tank 10
	    
	    "AI_Tank10_DB"(IB_Reset_PLC := "Total_DB".Restart_PLC,
	                  IB_Total_Reset := "Total_DB".Total_Reset_HMI,
	                  IB_EnablePowerControl := FALSE,
	                  IW_HW_UpLevel := 27648,
	                  IW_HW_LowLevel := 0,
	                  IW_Signal_from_Sensor := "IW_Tank10",
	                  IUDT_Analog_In := "UDT_AI_Tank10");
	    
	    "CalcVolume_Tank10_DB"(IW_ValueFromSensor := "AI_Tank10_DB".QDW_ScalledValue);
	    
	END_REGION
	
	REGION Bolgarska - Tank 1
	    
	    "AI_Tank11_DB"(IB_Reset_PLC := "Total_DB".Restart_PLC,
	                  IB_Total_Reset := "Total_DB".Total_Reset_HMI,
	                  IB_EnablePowerControl := FALSE,
	                  IW_HW_UpLevel := 27648,
	                  IW_HW_LowLevel := 0,
	                  IW_Signal_from_Sensor := "IW_Tank11",
	                  IUDT_Analog_In := "UDT_AI_Tank11");
	    
	    "CalcVolume_Tank11_DB"(IW_ValueFromSensor := "AI_Tank11_DB".QDW_ScalledValue);
	    
	END_REGION
	
	REGION Bolgarska - Tank 2
	    
	    "AI_Tank12_DB"(IB_Reset_PLC := "Total_DB".Restart_PLC,
	                  IB_Total_Reset := "Total_DB".Total_Reset_HMI,
	                  IB_EnablePowerControl := FALSE,
	                  IW_HW_UpLevel := 27648,
	                  IW_HW_LowLevel := 0,
	                  IW_Signal_from_Sensor := "IW_Tank12",
	                  IUDT_Analog_In := "UDT_AI_Tank12");
	    
	    "CalcVolume_Tank12_DB"(IW_ValueFromSensor := "AI_Tank12_DB".QDW_ScalledValue);
	    
	END_REGION
	
	REGION Bolgarska - Tank 3
	    
	    "AI_Tank13_DB"(IB_Reset_PLC := "Total_DB".Restart_PLC,
	                   IB_Total_Reset := "Total_DB".Total_Reset_HMI,
	                   IB_EnablePowerControl := FALSE,
	                   IW_HW_UpLevel := 27648,
	                   IW_HW_LowLevel := 0,
	                   IW_Signal_from_Sensor := "IW_Tank13", // Задати 
	                   IUDT_Analog_In := "UDT_AI_Tank13");
	    
	    "CalcVolume_Tank13_DB"(IW_ValueFromSensor := "AI_Tank13_DB".QDW_ScalledValue);
	    
	END_REGION
	
	REGION Bolgarska - Tank 4
	    
	    "AI_Tank14_DB"(IB_Reset_PLC := "Total_DB".Restart_PLC,
	                   IB_Total_Reset := "Total_DB".Total_Reset_HMI,
	                   IB_EnablePowerControl := FALSE,
	                   IW_HW_UpLevel := 27648,
	                   IW_HW_LowLevel := 0,
	                   IW_Signal_from_Sensor := "IW_Tank14", // Задати 
	                   IUDT_Analog_In := "UDT_AI_Tank14");
	    
	    "CalcVolume_Tank14_DB"(IW_ValueFromSensor := "AI_Tank14_DB".QDW_ScalledValue);
	    
	END_REGION
	
	
	
END_FUNCTION

ORGANIZATION_BLOCK "OB121"   // OB121, FBD, ProgrammingError
VERSION : 0.1
// stored: IsIECCheckEnabled false
   VAR_TEMP
      Temp_0 : Byte;
      Temp_1 : Byte;
      Temp_2 : Byte;
      Temp_3 : Byte;
      Temp_4 : Byte;
      Temp_5 : Byte;
      Temp_6 : Word;
      Temp_7 : Word;
      Temp_8 : Word;
      Temp_9 : Date_And_Time;
   END_VAR
BEGIN
END_ORGANIZATION_BLOCK

ORGANIZATION_BLOCK "OB122"   // OB122, FBD, IOAccessError
VERSION : 0.1
// stored: IsIECCheckEnabled false
   VAR_TEMP
      Temp_0 : Byte;
      Temp_1 : Byte;
      Temp_2 : Byte;
      Temp_3 : Byte;
      Temp_4 : Byte;
      Temp_5 : Byte;
      Temp_6 : Word;
      Temp_7 : Word;
      Temp_8 : Word;
      Temp_9 : Date_And_Time;
   END_VAR
BEGIN
END_ORGANIZATION_BLOCK

ORGANIZATION_BLOCK "OB80"   // OB80, FBD, TimeErrorInterrupt
VERSION : 0.1
// stored: IsIECCheckEnabled false
   VAR_TEMP
      Temp_0 : Byte;
      Temp_1 : Byte;
      Temp_2 : Byte;
      Temp_3 : Byte;
      Temp_4 : Byte;
      Temp_5 : Byte;
      Temp_6 : Word;
      Temp_7 : Byte;
      Temp_8 : Byte;
      Temp_9 : Byte;
      Temp_10 : Byte;
      Temp_11 : Date_And_Time;
   END_VAR
BEGIN
END_ORGANIZATION_BLOCK

ORGANIZATION_BLOCK "OB82"   // OB82, FBD, DiagnosticErrorInterrupt
VERSION : 0.1
// stored: IsIECCheckEnabled false
   VAR_TEMP
      Temp_0 : Byte;
      Temp_1 : Byte;
      Temp_2 : Byte;
      Temp_3 : Byte;
      Temp_4 : Byte;
      Temp_5 : Byte;
      Temp_6 : Word;
      Temp_7 : Bool;
      Temp_8 : Bool;
      Temp_9 : Bool;
      Temp_10 : Bool;
      Temp_11 : Bool;
      Temp_12 : Bool;
      Temp_13 : Bool;
      Temp_14 : Bool;
      Temp_15 : Byte;
      Temp_16 : Bool;
      Temp_17 : Bool;
      Temp_18 : Bool;
      Temp_19 : Bool;
      Temp_20 : Bool;
      Temp_21 : Bool;
      Temp_22 : Bool;
      Temp_23 : Bool;
      Temp_24 : Bool;
      Temp_25 : Bool;
      Temp_26 : Bool;
      Temp_27 : Bool;
      Temp_28 : Bool;
      Temp_29 : Bool;
      Temp_30 : Bool;
      Temp_31 : Bool;
      Temp_32 : Date_And_Time;
   END_VAR
BEGIN
END_ORGANIZATION_BLOCK

ORGANIZATION_BLOCK "OB83"   // OB83, FBD, PullOrPlugOfModules
VERSION : 0.1
// stored: IsIECCheckEnabled false
   VAR_TEMP
      Temp_0 : Byte;
      Temp_1 : Byte;
      Temp_2 : Byte;
      Temp_3 : Byte;
      Temp_4 : Byte;
      Temp_5 : Byte;
      Temp_6 : Word;
      Temp_7 : Int;
      Temp_8 : Word;
      Temp_9 : Date_And_Time;
   END_VAR
BEGIN
END_ORGANIZATION_BLOCK

ORGANIZATION_BLOCK "OB85"   // OB85, FBD, AccessError
VERSION : 0.1
// stored: IsIECCheckEnabled false
   VAR_TEMP
      Temp_0 : Byte;
      Temp_1 : Byte;
      Temp_2 : Byte;
      Temp_3 : Byte;
      Temp_4 : Byte;
      Temp_5 : Byte;
      Temp_6 : Int;
      Temp_7 : Byte;
      Temp_8 : Byte;
      Temp_9 : Byte;
      Temp_10 : Byte;
      Temp_11 : Date_And_Time;
   END_VAR
BEGIN
END_ORGANIZATION_BLOCK

ORGANIZATION_BLOCK "OB86"   // OB86, FBD, RackOrStationFailure
VERSION : 0.1
// stored: IsIECCheckEnabled false
   VAR_TEMP
      Temp_0 : Byte;
      Temp_1 : Byte;
      Temp_2 : Byte;
      Temp_3 : Byte;
      Temp_4 : Byte;
      Temp_5 : Byte;
      Temp_6 : Word;
      Temp_7 : Array[0..31] of Bool;
      Temp_8 : Date_And_Time;
   END_VAR
BEGIN
END_ORGANIZATION_BLOCK

ORGANIZATION_BLOCK "OB87"   // OB87, FBD, CommunicationError
VERSION : 0.1
// stored: IsIECCheckEnabled false
   VAR_TEMP
      Temp_0 : Byte;
      Temp_1 : Byte;
      Temp_2 : Byte;
      Temp_3 : Byte;
      Temp_4 : Byte;
      Temp_5 : Byte;
      Temp_6 : Word;
      Temp_7 : DWord;
      Temp_8 : Date_And_Time;
   END_VAR
BEGIN
END_ORGANIZATION_BLOCK

FUNCTION "FC_Scale_Instance" : Void   // FC19, FBD
VERSION : 0.1
// stored: AutoNumber true, IsIECCheckEnabled false, UDAEnableTagReadback false
BEGIN

REGION Network 1
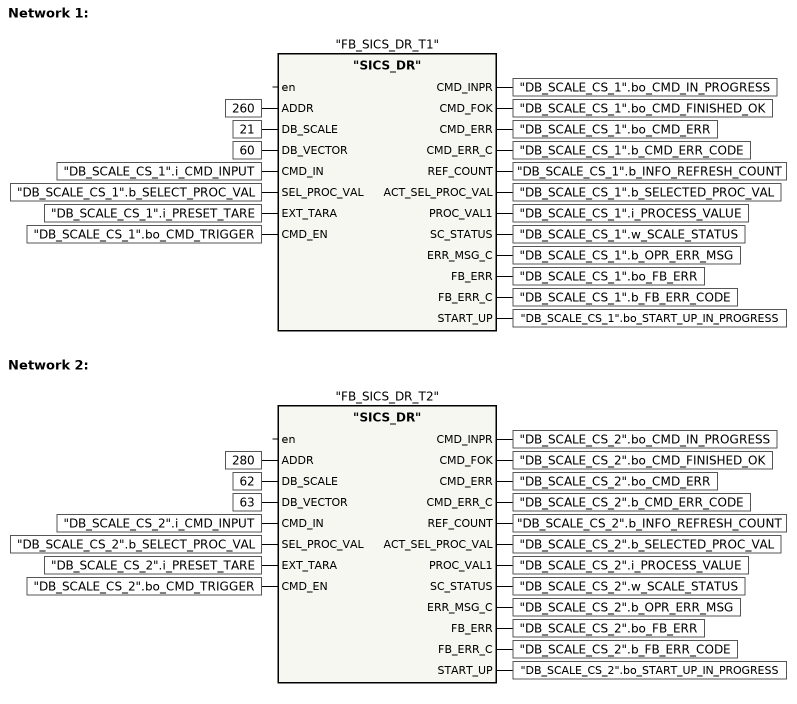
   "FB_SICS_DR_T1"(ADDR := 260,   // "SICS_DR"
                   DB_SCALE := 21,
                   DB_VECTOR := 60,
                   CMD_IN := "DB_SCALE_CS_1".i_CMD_INPUT,
                   SEL_PROC_VAL := "DB_SCALE_CS_1".b_SELECT_PROC_VAL,
                   EXT_TARA := "DB_SCALE_CS_1".i_PRESET_TARE,
                   CMD_EN := "DB_SCALE_CS_1".bo_CMD_TRIGGER,
                   CMD_INPR => "DB_SCALE_CS_1".bo_CMD_IN_PROGRESS,
                   CMD_FOK => "DB_SCALE_CS_1".bo_CMD_FINISHED_OK,
                   CMD_ERR => "DB_SCALE_CS_1".bo_CMD_ERR,
                   CMD_ERR_C => "DB_SCALE_CS_1".b_CMD_ERR_CODE,
                   REF_COUNT => "DB_SCALE_CS_1".b_INFO_REFRESH_COUNT,
                   ACT_SEL_PROC_VAL => "DB_SCALE_CS_1".b_SELECTED_PROC_VAL,
                   PROC_VAL1 => "DB_SCALE_CS_1".i_PROCESS_VALUE,
                   SC_STATUS => "DB_SCALE_CS_1".w_SCALE_STATUS,
                   ERR_MSG_C => "DB_SCALE_CS_1".b_OPR_ERR_MSG,
                   FB_ERR => "DB_SCALE_CS_1".bo_FB_ERR,
                   FB_ERR_C => "DB_SCALE_CS_1".b_FB_ERR_CODE,
                   START_UP => "DB_SCALE_CS_1".bo_START_UP_IN_PROGRESS);
END_REGION

REGION Network 2
   "FB_SICS_DR_T2"(ADDR := 280,   // "SICS_DR"
                   DB_SCALE := 62,
                   DB_VECTOR := 63,
                   CMD_IN := "DB_SCALE_CS_2".i_CMD_INPUT,
                   SEL_PROC_VAL := "DB_SCALE_CS_2".b_SELECT_PROC_VAL,
                   EXT_TARA := "DB_SCALE_CS_2".i_PRESET_TARE,
                   CMD_EN := "DB_SCALE_CS_2".bo_CMD_TRIGGER,
                   CMD_INPR => "DB_SCALE_CS_2".bo_CMD_IN_PROGRESS,
                   CMD_FOK => "DB_SCALE_CS_2".bo_CMD_FINISHED_OK,
                   CMD_ERR => "DB_SCALE_CS_2".bo_CMD_ERR,
                   CMD_ERR_C => "DB_SCALE_CS_2".b_CMD_ERR_CODE,
                   REF_COUNT => "DB_SCALE_CS_2".b_INFO_REFRESH_COUNT,
                   ACT_SEL_PROC_VAL => "DB_SCALE_CS_2".b_SELECTED_PROC_VAL,
                   PROC_VAL1 => "DB_SCALE_CS_2".i_PROCESS_VALUE,
                   SC_STATUS => "DB_SCALE_CS_2".w_SCALE_STATUS,
                   ERR_MSG_C => "DB_SCALE_CS_2".b_OPR_ERR_MSG,
                   FB_ERR => "DB_SCALE_CS_2".bo_FB_ERR,
                   FB_ERR_C => "DB_SCALE_CS_2".b_FB_ERR_CODE,
                   START_UP => "DB_SCALE_CS_2".bo_START_UP_IN_PROGRESS);
END_REGION
END_FUNCTION

FUNCTION "FC_Scale_Mng" : Void   // FC19, FBD
VERSION : 0.1
// stored: AutoNumber true, IsIECCheckEnabled false, UDAEnableTagReadback false
BEGIN

REGION Network 1
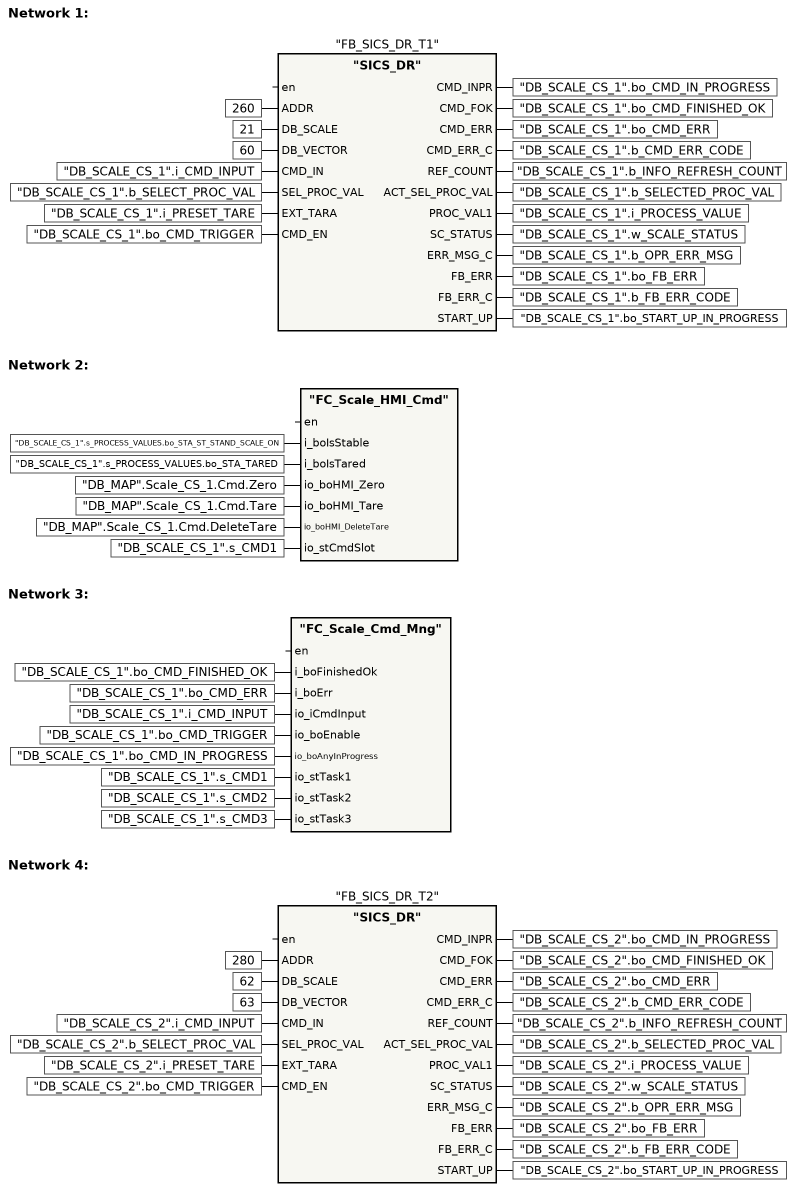
   "FB_SICS_DR_T1"(ADDR := 260,   // "SICS_DR"
                   DB_SCALE := 21,
                   DB_VECTOR := 60,
                   CMD_IN := "DB_SCALE_CS_1".i_CMD_INPUT,
                   SEL_PROC_VAL := "DB_SCALE_CS_1".b_SELECT_PROC_VAL,
                   EXT_TARA := "DB_SCALE_CS_1".i_PRESET_TARE,
                   CMD_EN := "DB_SCALE_CS_1".bo_CMD_TRIGGER,
                   CMD_INPR => "DB_SCALE_CS_1".bo_CMD_IN_PROGRESS,
                   CMD_FOK => "DB_SCALE_CS_1".bo_CMD_FINISHED_OK,
                   CMD_ERR => "DB_SCALE_CS_1".bo_CMD_ERR,
                   CMD_ERR_C => "DB_SCALE_CS_1".b_CMD_ERR_CODE,
                   REF_COUNT => "DB_SCALE_CS_1".b_INFO_REFRESH_COUNT,
                   ACT_SEL_PROC_VAL => "DB_SCALE_CS_1".b_SELECTED_PROC_VAL,
                   PROC_VAL1 => "DB_SCALE_CS_1".i_PROCESS_VALUE,
                   SC_STATUS => "DB_SCALE_CS_1".w_SCALE_STATUS,
                   ERR_MSG_C => "DB_SCALE_CS_1".b_OPR_ERR_MSG,
                   FB_ERR => "DB_SCALE_CS_1".bo_FB_ERR,
                   FB_ERR_C => "DB_SCALE_CS_1".b_FB_ERR_CODE,
                   START_UP => "DB_SCALE_CS_1".bo_START_UP_IN_PROGRESS);
END_REGION

REGION Network 2
   "FC_Scale_HMI_Cmd"(i_boIsStable := "DB_SCALE_CS_1".s_PROCESS_VALUES.bo_STA_ST_STAND_SCALE_ON,
                      i_boIsTared := "DB_SCALE_CS_1".s_PROCESS_VALUES.bo_STA_TARED,
                      io_boHMI_Zero := "DB_MAP".Scale_CS_1.Cmd.Zero,
                      io_boHMI_Tare := "DB_MAP".Scale_CS_1.Cmd.Tare,
                      io_boHMI_DeleteTare := "DB_MAP".Scale_CS_1.Cmd.DeleteTare,
                      io_stCmdSlot := "DB_SCALE_CS_1".s_CMD1);
END_REGION

REGION Network 3
   "FC_Scale_Cmd_Mng"(i_boFinishedOk := "DB_SCALE_CS_1".bo_CMD_FINISHED_OK,
                      i_boErr := "DB_SCALE_CS_1".bo_CMD_ERR,
                      io_iCmdInput := "DB_SCALE_CS_1".i_CMD_INPUT,
                      io_boEnable := "DB_SCALE_CS_1".bo_CMD_TRIGGER,
                      io_boAnyInProgress := "DB_SCALE_CS_1".bo_CMD_IN_PROGRESS,
                      io_stTask1 := "DB_SCALE_CS_1".s_CMD1,
                      io_stTask2 := "DB_SCALE_CS_1".s_CMD2,
                      io_stTask3 := "DB_SCALE_CS_1".s_CMD3);
END_REGION

REGION Network 4
   "FB_SICS_DR_T2"(ADDR := 280,   // "SICS_DR"
                   DB_SCALE := 62,
                   DB_VECTOR := 63,
                   CMD_IN := "DB_SCALE_CS_2".i_CMD_INPUT,
                   SEL_PROC_VAL := "DB_SCALE_CS_2".b_SELECT_PROC_VAL,
                   EXT_TARA := "DB_SCALE_CS_2".i_PRESET_TARE,
                   CMD_EN := "DB_SCALE_CS_2".bo_CMD_TRIGGER,
                   CMD_INPR => "DB_SCALE_CS_2".bo_CMD_IN_PROGRESS,
                   CMD_FOK => "DB_SCALE_CS_2".bo_CMD_FINISHED_OK,
                   CMD_ERR => "DB_SCALE_CS_2".bo_CMD_ERR,
                   CMD_ERR_C => "DB_SCALE_CS_2".b_CMD_ERR_CODE,
                   REF_COUNT => "DB_SCALE_CS_2".b_INFO_REFRESH_COUNT,
                   ACT_SEL_PROC_VAL => "DB_SCALE_CS_2".b_SELECTED_PROC_VAL,
                   PROC_VAL1 => "DB_SCALE_CS_2".i_PROCESS_VALUE,
                   SC_STATUS => "DB_SCALE_CS_2".w_SCALE_STATUS,
                   ERR_MSG_C => "DB_SCALE_CS_2".b_OPR_ERR_MSG,
                   FB_ERR => "DB_SCALE_CS_2".bo_FB_ERR,
                   FB_ERR_C => "DB_SCALE_CS_2".b_FB_ERR_CODE,
                   START_UP => "DB_SCALE_CS_2".bo_START_UP_IN_PROGRESS);
END_REGION

REGION Network 5
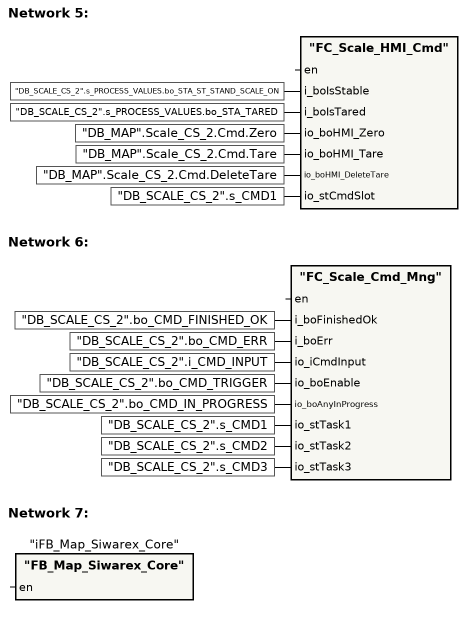
   "FC_Scale_HMI_Cmd"(i_boIsStable := "DB_SCALE_CS_2".s_PROCESS_VALUES.bo_STA_ST_STAND_SCALE_ON,
                      i_boIsTared := "DB_SCALE_CS_2".s_PROCESS_VALUES.bo_STA_TARED,
                      io_boHMI_Zero := "DB_MAP".Scale_CS_2.Cmd.Zero,
                      io_boHMI_Tare := "DB_MAP".Scale_CS_2.Cmd.Tare,
                      io_boHMI_DeleteTare := "DB_MAP".Scale_CS_2.Cmd.DeleteTare,
                      io_stCmdSlot := "DB_SCALE_CS_2".s_CMD1);
END_REGION

REGION Network 6
   "FC_Scale_Cmd_Mng"(i_boFinishedOk := "DB_SCALE_CS_2".bo_CMD_FINISHED_OK,
                      i_boErr := "DB_SCALE_CS_2".bo_CMD_ERR,
                      io_iCmdInput := "DB_SCALE_CS_2".i_CMD_INPUT,
                      io_boEnable := "DB_SCALE_CS_2".bo_CMD_TRIGGER,
                      io_boAnyInProgress := "DB_SCALE_CS_2".bo_CMD_IN_PROGRESS,
                      io_stTask1 := "DB_SCALE_CS_2".s_CMD1,
                      io_stTask2 := "DB_SCALE_CS_2".s_CMD2,
                      io_stTask3 := "DB_SCALE_CS_2".s_CMD3);
END_REGION

REGION Network 7
   "iFB_Map_Siwarex_Core"();   // "FB_Map_Siwarex_Core"
END_REGION
END_FUNCTION

FUNCTION "FC_Scale_HMI_Cmd" : Void
{ S7_Optimized_Access := 'FALSE' }
VERSION : 1.2
   VAR_INPUT 
      i_boIsStable : Bool;   // Статус модуля: Весы стабильны (Standstill)
      i_boIsTared : Bool;   // Статус модуля: Весы затарированы
   END_VAR

   VAR_IN_OUT 
      io_boHMI_Zero : Bool;   // Кнопка HMI: Обнулить
      io_boHMI_Tare : Bool;   // Кнопка HMI: Затарировать
      io_boHMI_DeleteTare : Bool;   // Кнопка HMI: Удалить тару
      io_stCmdSlot : "UDT_SIWA_Cmd";   // Слот задачи для передачи в менеджер (напр. sTask2)
   END_VAR


BEGIN
	    // =========================================================
	    // 1. Обнуление (Код 21)
	    // =========================================================
	    IF #io_boHMI_Zero THEN
	        IF #i_boIsStable AND NOT #io_stCmdSlot.bo_InProgress THEN
	            #io_stCmdSlot.i_Code := 21;
	            #io_stCmdSlot.bo_Trigger := TRUE;
	        END_IF;
	        #io_boHMI_Zero := FALSE;
	    END_IF;
	    
	    // =========================================================
	    // 2. Тарирование (Код 22)
	    // Защита от двойной тары (NOT i_boIsTared)
	    // =========================================================
	    IF #io_boHMI_Tare THEN
	        IF #i_boIsStable AND NOT #i_boIsTared AND NOT #io_stCmdSlot.bo_InProgress THEN
	            #io_stCmdSlot.i_Code := 22;
	            #io_stCmdSlot.bo_Trigger := TRUE;
	        END_IF;
	        #io_boHMI_Tare := FALSE;
	    END_IF;
	    
	    // =========================================================
	    // 3. Удаление тары (Код 24)
	    // =========================================================
	    IF #io_boHMI_DeleteTare THEN
	        IF #i_boIsTared AND NOT #io_stCmdSlot.bo_InProgress THEN
	            #io_stCmdSlot.i_Code := 24;
	            #io_stCmdSlot.bo_Trigger := TRUE;
	        END_IF;
	        #io_boHMI_DeleteTare := FALSE;
	    END_IF;
	    
END_FUNCTION

FUNCTION "FC_Scale_Cmd_Mng" : Void
{ S7_Optimized_Access := 'FALSE' }
VERSION : 1.6
   VAR_INPUT 
      i_boFinishedOk : Bool;   // Аппаратный статус: Команда завершена успешно
      i_boErr : Bool;   // Аппаратный статус: Ошибка выполнения
   END_VAR

   VAR_IN_OUT 
      io_iCmdInput : Int;   // Регистр команды модуля Siwarex
      io_boEnable : Bool;   // Триггер запуска аппаратной команды
      io_boAnyInProgress : Bool;   // Флаг: Модуль занят
      io_stTask1 : "UDT_SIWA_Cmd";   // Слот 1 (Высокий приоритет, напр. HMI)
      io_stTask2 : "UDT_SIWA_Cmd";   // Слот 2
      io_stTask3 : "UDT_SIWA_Cmd";   // Слот 3 (Низкий приоритет, напр. DR30)
   END_VAR


BEGIN
	    // 1. Очистка импульсных статусов
	    #io_stTask1.bo_FinishedOk := FALSE;
	    #io_stTask1.bo_FinishedError := FALSE;
	    
	    #io_stTask2.bo_FinishedOk := FALSE;
	    #io_stTask2.bo_FinishedError := FALSE;
	    
	    #io_stTask3.bo_FinishedOk := FALSE;
	    #io_stTask3.bo_FinishedError := FALSE;
	    
	    // 2. Проверка завершения текущей задачи
	    IF #io_boAnyInProgress THEN
	        IF #io_stTask1.bo_InProgress THEN
	            IF #i_boFinishedOk THEN
	                #io_stTask1.bo_FinishedOk := TRUE;
	            END_IF;
	            IF #i_boErr THEN
	                #io_stTask1.bo_FinishedError := TRUE;
	            END_IF;
	            
